// TwinCAT 3 PLC project OC_Profinet
// Title: OC_Profinet
// Company: Open Commissioning
// Author: SpiraTec AG
// ProjectVersion: 1.0.1
// Description: Open Commissioning Library for Profinet devices
// ProgramVersion: 3.1.4026.19
// libraries:
//   OC_Core, * (Open Commissioning)
//   OC_Profisafe, * (Open Commissioning)
//   Tc2_Math, * (Beckhoff Automation GmbH)
//   Tc2_Standard, * (Beckhoff Automation GmbH)
//   Tc2_System, * (Beckhoff Automation GmbH)
//   Tc2_Utilities, * (Beckhoff Automation GmbH)
//   Tc3_Module, * (Beckhoff Automation GmbH)
//   TcUnit, * (www.tcunit.org)
// project tree:
//   Common/ProfidriveGSM/ E_ProfidriveGSM_State.TcTLEO, FB_ProfidriveGSM.TcPOU, ST_ProfidriveGSM_Control.TcDUT, ST_ProfidriveGSM_Status.TcDUT
//   Common/ProfidriveParamInterpreter/ E_ProfidriveParam_Format.TcDUT, FB_ProfidriveParamInterpreter.TcPOU, ST_ProfidriveParam.TcDUT, ST_ProfidriveParam_Set.TcDUT
//   Common/Utils/ F_CalcCrc16.TcPOU
//   Devices/ I_SEW_Movisafe.TcIO
//   Devices/Profidrive_Telegram1/ FB_Profidrive_Telegram1.TcPOU, ST_Profidrive_Telegram1_Config.TcDUT, ST_Profidrive_Telegram1_Control.TcDUT, ST_Profidrive_Telegram1_Status.TcDUT
//   Devices/Siemens_RcvDp/ FB_Siemens_RcvDp.TcPOU, ST_Siemens_RcvDp_Config.TcDUT, ST_Siemens_RcvDp_Control.TcDUT, ST_Siemens_RcvDp_DevData.TcDUT, ST_Siemens_RcvDp_HstData.TcDUT, ST_Siemens_RcvDp_Status.TcDUT
//   Devices/Siemens_SendDp/ FB_Siemens_SendDp.TcPOU, ST_Siemens_SendDp_Config.TcDUT, ST_Siemens_SendDp_Control.TcDUT, ST_Siemens_SendDp_DevData.TcDUT, ST_Siemens_SendDp_HstData.TcDUT, ST_Siemens_SendDp_Status.TcDUT
//   Devices/SEW_MoviC_Position/ E_SEW_MoviC_Position_OperationMode.TcDUT, FB_SEW_MoviC_Position.TcPOU, ST_SEW_MoviC_Position_Config.TcDUT, ST_SEW_MoviC_Position_Control.TcDUT, ST_SEW_MoviC_Position_Status.TcDUT
//   Devices/SEW_MoviC_Velocity/ FB_SEW_MoviC_Velocity.TcPOU, ST_SEW_MoviC_Velocity_Config.TcDUT, ST_SEW_MoviC_Velocity_Control.TcDUT, ST_SEW_MoviC_Velocity_Status.TcDUT
//   Devices/SEW_Movisafe_CSSx1a/ FB_SEW_Movisafe_CSSx1a.TcPOU, ST_SEW_Movisafe_CSSx1a_Config.TcDUT, ST_SEW_Movisafe_CSSx1a_Control.TcDUT, ST_SEW_Movisafe_CSSx1a_Status.TcDUT
//   / PlcTask.TcTTO
//   Tests/Devices/ FB_ProfidriveGSM_Test.TcPOU, FB_ProfidriveTelegram1_Test.TcPOU, FB_SEW_MoviC_Position_Test.TcPOU, FB_SEW_MoviC_Velocity_Test.TcPOU, FB_Siemens_RcvDp_Test.TcPOU, FB_SEW_Movisafe_CSSx1a_Test.TcPOU, FB_Siemens_SendDp_Test.TcPOU
//   Tests/Helpers/ FB_SEW_Movisafe.TcPOU
//   Tests/ PRG_TEST.TcPOU
//   _backlog/Danfoss_VLT_MCA_120/ FB_Danfoss_VLT_MCA_120.TcPOU, ST_Danfoss_VLT_MCA_120_Config.TcDUT, ST_Danfoss_VLT_MCA_120_Control.TcDUT, ST_Danfoss_VLT_MCA_120_Status.TcDUT (not stored)
//   _backlog/ProfidriveCu/ FB_ProfidriveCu.TcPOU, I_Sinamics.TcIO (not stored), ST_ProfidriveCuConfig.TcDUT (not stored)
//   _backlog/SEW_Movisafe_CSBx1a/ FB_SEW_Movisafe_CSBx1a.TcPOU, ST_SEW_Movisafe_CSBx1a_Config.TcDUT, ST_SEW_Movisafe_CSBx1a_Control.TcDUT, ST_SEW_Movisafe_CSBx1a_Status.TcDUT

CONFIGURATION OC_Profinet
    RESOURCE PLC ON TwinCAT3
        TASK PlcTask(INTERVAL := T#1ms, PRIORITY := 6);
        PROGRAM PRG_TEST WITH PlcTask : PRG_TEST;
    END_RESOURCE
END_CONFIGURATION

// ---- Common/ProfidriveGSM/E_ProfidriveGSM_State.TcTLEO
{attribute 'qualified_only'}
{attribute 'strict'}
{attribute 'conditionalshow'}
TYPE E_ProfidriveGSM_State :
(
	S0_Disabled := 0,
	S1_SwitchingOnInhibited := 1,
	S2_ReadyForSwitchingOn := 2,
	S3_SwitchedOn := 3,
	S4_Operation := 4,
	S51_RampStop := 51,
	S52_QuickStop := 52
);
END_TYPE

// ---- Common/ProfidriveGSM/ST_ProfidriveGSM_Control.TcDUT
(*
	Steuerwort 1 (STW1)
	Steuerwort 1 SIEMENS Telegramm 10x
	https://cache.industry.siemens.com/dl/files/665/109770665/att_1023132/v2/109770665_PROFIdrive_Statemachine_DOC_V10_de.pdf
*)
{attribute 'pack_mode' := '1'}
TYPE ST_ProfidriveGSM_Control :
STRUCT
	b0_On 							: BIT; 	//ON/OFF (OFF1)
	b1_CoastStop					: BIT; 	//The axis will not coast stop if this bit is set (OFF2)
	b2_QuickStop					: BIT; 	//The axis will not execute quick stop if this bit is set. Quick stop executes a controlled stop on the axis. (OFF3)
	b3_EnableOperation				: BIT; 	//The axis will enable and execute command if all preconditions are set. If a Wake and Shake procedure has to be executed as part of enabling, the transition to state "S4: Operation Enabled" is delayed until the procedure is finished.
	b4_Reserve						: BIT;	//Reserve
	b5_Reserve						: BIT;	//Reserve
	b6_Reserve						: BIT;	//Reserve
	b7_FaultAcknowledge				: BIT;	//Set this bit to reset faults on the drive.
	b8_Reserve						: BIT;	//Reserve
	b9_Reserve						: BIT;	//Reserve	
	b10_ControlPlc					: BIT;	//When not set, no command is accepted from the PLC.	
	b11_Reserved					: BIT;	//Reserve
	b12_Reserved					: BIT;	//Reserve
	b13_Reserved					: BIT;	//Reserve
	b14_Reserved					: BIT;	//Reserve
	b15_Reserved					: BIT;	//Reserve
END_STRUCT
END_TYPE

// ---- Common/ProfidriveGSM/ST_ProfidriveGSM_Status.TcDUT
(*
	Zustandswort 1 (ZSW1)
	Zustandswort 1 SIEMENS Telegramm 10x
	https://cache.industry.siemens.com/dl/files/665/109770665/att_1023132/v2/109770665_PROFIdrive_Statemachine_DOC_V10_de.pdf
*)

{attribute 'pack_mode' := '1'}
TYPE ST_ProfidriveGSM_Status :
STRUCT
	b0_ReadyToSwitchOn 				: BIT; 	//Ready to switch on
	b1_ReadyForOperation			: BIT; 	//Ready for operation
	b2_OperationEnabled				: BIT; 	//Operation enabled
	b3_FaultPresent					: BIT; 	//A fault is present on the axis
	b4_CoastStop 					: BIT;	//No coast stop is executed (No OFF2 is active)
	b5_QuickStop					: BIT;	//No quick stop is executed (No OFF3 is active)
	b6_SwitchingOnInhibited			: BIT;	//Switch-on inhibit Switching on again is only possible through OFF1 and subsequent ON.
	b7_WarningPresent				: BIT;	//Warning present. The drive is operating. No acknowledgment required
	b8_Reserve						: BIT;	//Reserve
	b9_ControlRequested				: BIT;	//Control requested by the master
	b10_Reserved					: BIT;	//Reserve
	b11_Reserved					: BIT;	//Reserve
	b12_Reserved					: BIT;	//Reserve
	b13_Reserved					: BIT;	//Reserve
	b14_Reserved					: BIT;	//Reserve
	b15_Reserved					: BIT;	//Reserve
END_STRUCT
END_TYPE

// ---- Common/ProfidriveParamInterpreter/E_ProfidriveParam_Format.TcDUT
{attribute 'qualified_only'}
{attribute 'strict'}
{attribute 'conditionalshow'}
TYPE E_ProfidriveParam_Format :
(
	UNKNOWN := 0,
	INT8	:= 2,
	INT16	:= 3,
	INT32	:= 4,
	UINT8	:= 5,
	UINT16	:= 6,
	UINT32	:= 7,
	FLOAT	:= 8,
	ZERO	:= 64,
	BYTE_	:= 65,
	WORD_	:= 66,
	DWORD_	:= 67,
	ERROR	:= 68
) BYTE;
END_TYPE

// ---- Common/ProfidriveParamInterpreter/ST_ProfidriveParam.TcDUT
{attribute 'conditionalshow'}
TYPE ST_ProfidriveParam :
STRUCT
	nAttribute	: BYTE;
	nNumber		: UINT;
	nSubIndex	: UINT;
	nElements	: BYTE;
	nFormat		: E_ProfidriveParam_Format;
	aValue		: ARRAY[0..234] OF BYTE;
END_STRUCT
END_TYPE

// ---- Common/ProfidriveParamInterpreter/ST_ProfidriveParam_Set.TcDUT
{attribute 'conditionalshow'}
TYPE ST_ProfidriveParam_Set :
	ARRAY[0..22] OF ST_ProfidriveParam; 
END_TYPE

// ---- Devices/Profidrive_Telegram1/ST_Profidrive_Telegram1_Config.TcDUT
TYPE ST_Profidrive_Telegram1_Config :
STRUCT
	bForceMode					: BOOL; //Ignore process data from fieldbus.
	bSwapProcessData			: BOOL; //Reverse process data byte order from/to fieldbus.
	fRampDownTimeCoastStop 		: REAL := 1.0;		//Coast stop deceleration time in s
	bControlRequested			: BOOL := TRUE;
	bOutputVelocity				: BOOL := TRUE;		//TRUE: TargetValue = Velocity, FALSE: TargetValue = Position
	fP1058						: REAL := 150.0;	//JOG 1 velocity in rotation/s
	fP1059						: REAL := -150.0;	//JOG 1 velocity in rotation/s
	fP1120						: REAL := 2.0;		//Default acceleration time in s
	fP1121						: REAL := 2.0;		//Default deceleration time in s
	fP1135						: REAL := 1.0;		//Ramp down time quick stop in s
	fP2000						: REAL := 3000;		//Velocity in rotation/s when targeting 16#4000
	nR0035						: REAL := 60.0; 	//Temperature in degree celcius	
END_STRUCT
END_TYPE

// ---- Devices/Profidrive_Telegram1/ST_Profidrive_Telegram1_Control.TcDUT
TYPE ST_Profidrive_Telegram1_Control :
STRUCT
	b0_Off1								: BOOL;	//STW1_0	0 = OFF1 (braking with ramp-function generator, then pulse suppression & ready for switching on) | 0 → 1 = ON (pulses can be enabled)
	b1_Off2								: BOOL;	//STW1_1	0 = OFF2 (immediate pulse suppression and switching on inhibited) | 1 = No OFF2 (enable is possible)
	b2_Off3								: BOOL;	//STW1_2	0 = OFF3 (braking with the OFF3 ramp p1135, then pulse suppression and switching on inhibited) | 1 = No OFF3 (enable possible) 
	b3_EnableOperation					: BOOL;	//STW1_3	0 = Inhibit operation (suppress pulses) | 1 = Enable operation (pulses can be enabled) 
	b4_OperatingCondition				: BOOL;	//STW1_4	0 = Inhibit ramp-function generator (set the ramp-function generator output to zero) | 1 = Operating condition (the ramp-function generator can be enabled)
	b5_ContinueRampFunctionGenerator	: BOOL;	//STW1_5	0 = Freeze ramp-function generator (freeze the ramp-function generator output) | 1 = Continue ramp-function generator 
	b6_EnableSetpoint  					: BOOL;	//STW1_6	0 = Inhibit setpoint (set the ramp-function generator input to zero) | 1 = Enable setpoint 
	b7_AcknowledgeFaults				: BOOL;	//STW1_7	0 → 1: = Acknowledge faults	                            
	b8_Jog1								: BOOL;	//STW1_8	1 = Jog 1 signal source
	b9_Jog2								: BOOL;	//STW1_9	1 = Jog 2 signal source
	b10_ControlByPlc					: BOOL;	//STW1_10	1 = Control by PLC
	b11_SetpointInversion				: BOOL;	//STW1_11	1 = Setpoint inversion
	b12_Reserved						: BOOL;	//STW1_12	Reserved
	b13_PotentiometerSetpointRaise		: BOOL;	//STW1_13	1 = Motorized potentiometer setpoint raise
	b14_PotentiometerSetpointLower		: BOOL;	//STW1_14	1 = Motorized potentiometer setpoint lower
	b15_Reserved						: BOOL;	//STW1_15	Reserved	
	nTargetVelocity						: INT;
END_STRUCT
END_TYPE

// ---- Devices/Profidrive_Telegram1/ST_Profidrive_Telegram1_Status.TcDUT
TYPE ST_Profidrive_Telegram1_Status :
STRUCT
	b0_ReadyForSwitchingOn				: BOOL; // ZSW1_0	1 = Ready for switching on
	b1_ReadyForOperation				: BOOL; // ZSW1_1	1 = Ready for operation
	b2_OperationEnabled					: BOOL; // ZSW1_2	1 = Operation enabled
	b3_FaultPresent						: BOOL; // ZSW1_3	1 = Fault present
	b4_NoCoastDownActive				: BOOL; // ZSW1_4	1 = No coast down active (OFF2 inactive)
	b5_NoQuickStopActive				: BOOL; // ZSW1_5	1 = No quick stop active (OFF3 inactive)
	b6_SwitchingOnInhibited				: BOOL; // ZSW1_6	1 = Switching on inhibited active
	b7_AlarmPresent						: BOOL; // ZSW1_7	1 = Alarm present                        	
	b8_DeviationWithinTolerance			: BOOL; // ZSW1_8	1 = Speed setpoint - actual value deviation within tolerance t_off
	b9_ControlRequested					: BOOL; // ZSW1_9	1 = Control requested        
	b10_RpmCompValueReachedOrExceeded	: BOOL; // ZSW1_10	1 = f or n comparison value reached/exceeded  
	b11_TorqueOrPowerLimitNotReached	: BOOL; // ZSW1_11	1 = I, M, or P limit not reached     
	b12_OpenHoldingBrake 				: BOOL; // ZSW1_12	1 = Open the holding brake      
	b13_NoOvertempAlarm					: BOOL; // ZSW1_13	1 = No motor overtemperature alarm      
	b14_MotorRotatesForwards			: BOOL; // ZSW1_14	1 = Motor rotates forwards (n_act >= 0) | 0 = Motor rotates backwards (n_act < 0)   
	b15_NoAlarmNoOvertempPowerUnit		: BOOL; // ZSW1_15	1 = No alarm, thermal overload, power unit  
	nVelocity							: INT;
END_STRUCT
END_TYPE

// ---- Devices/Siemens_RcvDp/ST_Siemens_RcvDp_Config.TcDUT
TYPE ST_Siemens_RcvDp_Config :
STRUCT
	bForceMode			: BOOL; //Ignore process data from fieldbus.
	bSwapProcessData	: BOOL; //Reverse process data byte order from/to fieldbus.
	nDpDpId			 	: UINT := 0;
	fTimeout		 	: REAL := 0.5;
	bAutoAckRei			: BOOL := TRUE;
END_STRUCT
END_TYPE

// ---- Devices/Siemens_RcvDp/ST_Siemens_RcvDp_Control.TcDUT
{attribute 'pack_mode' := '1'}
TYPE ST_Siemens_RcvDp_Control :
STRUCT
	nRcvBoolData			: WORD;
	nRcvInt00				: INT;
	nRcvInt01				: INT;
	nRcvData				: WORD;
	nRcvSequenceNumber		: WORD;
	nRcvCrc					: WORD;
END_STRUCT
END_TYPE

// ---- Devices/Siemens_RcvDp/ST_Siemens_RcvDp_DevData.TcDUT
TYPE ST_Siemens_RcvDp_DevData :
STRUCT
	bAckRei		: BOOL;
	bSub00		: BOOL;
	bSub01		: BOOL;
	bSub02		: BOOL;
	bSub03		: BOOL;
	bSub04		: BOOL;
	bSub05		: BOOL;
	bSub06		: BOOL;
	bSub07		: BOOL;
	bSub08		: BOOL;
	bSub09		: BOOL;
	bSub10		: BOOL;
	bSub11		: BOOL;
	bSub12		: BOOL;
	bSub13		: BOOL;
	bSub14		: BOOL;
	bSub15		: BOOL;
	nSub00		: INT;
	nSub01		: INT;
END_STRUCT
END_TYPE

// ---- Devices/Siemens_RcvDp/ST_Siemens_RcvDp_HstData.TcDUT
TYPE ST_Siemens_RcvDp_HstData :
STRUCT
	bError		: BOOL;
	bSubsOn		: BOOL;
	bRcv00		: BOOL;
	bRcv01		: BOOL;
	bRcv02		: BOOL;
	bRcv03		: BOOL;
	bRcv04		: BOOL;
	bRcv05		: BOOL;
	bRcv06		: BOOL;
	bRcv07		: BOOL;
	bRcv08		: BOOL;
	bRcv09		: BOOL;
	bRcv10		: BOOL;
	bRcv11		: BOOL;
	bRcv12		: BOOL;
	bRcv13		: BOOL;
	bRcv14		: BOOL;
	bRcv15		: BOOL;
	nRcv00		: INT;
	nRcv01		: INT;
END_STRUCT
END_TYPE

// ---- Devices/Siemens_RcvDp/ST_Siemens_RcvDp_Status.TcDUT
{attribute 'pack_mode' := '1'}
TYPE ST_Siemens_RcvDp_Status :
STRUCT
	nSendData				: WORD;
	nSendSequenceNumber		: WORD;	
	nSendCrc				: WORD;
END_STRUCT
END_TYPE

// ---- Devices/Siemens_SendDp/ST_Siemens_SendDp_Config.TcDUT
TYPE ST_Siemens_SendDp_Config :
STRUCT
	bForceMode			: BOOL; //Ignore process data from fieldbus.
	bSwapProcessData	: BOOL; //Reverse process data byte order from/to fieldbus.
	nDpDpId			 	: UINT := 0;
	fTimeout		 	: REAL := 0.5;
END_STRUCT
END_TYPE

// ---- Devices/Siemens_SendDp/ST_Siemens_SendDp_Control.TcDUT
TYPE ST_Siemens_SendDp_Control :
STRUCT
	nRcvData				: WORD;
	nRcvSequenceNumber		: WORD;	
	nRcvCrc					: WORD;
END_STRUCT
END_TYPE

// ---- Devices/Siemens_SendDp/ST_Siemens_SendDp_DevData.TcDUT
TYPE ST_Siemens_SendDp_DevData :
STRUCT
	bSend00		: BOOL;
	bSend01		: BOOL;
	bSend02		: BOOL;
	bSend03		: BOOL;
	bSend04		: BOOL;
	bSend05		: BOOL;
	bSend06		: BOOL;
	bSend07		: BOOL;
	bSend08		: BOOL;
	bSend09		: BOOL;
	bSend10		: BOOL;
	bSend11		: BOOL;
	bSend12		: BOOL;
	bSend13		: BOOL;
	bSend14		: BOOL;
	bSend15		: BOOL;
	nSend00		: INT;
	nSend01		: INT;
END_STRUCT
END_TYPE

// ---- Devices/Siemens_SendDp/ST_Siemens_SendDp_HstData.TcDUT
TYPE ST_Siemens_SendDp_HstData :
STRUCT
	bError		: BOOL;
	bSubsOn		: BOOL;
END_STRUCT
END_TYPE

// ---- Devices/Siemens_SendDp/ST_Siemens_SendDp_Status.TcDUT
TYPE ST_Siemens_SendDp_Status :
STRUCT
	nSendBoolData			: WORD;
	nSendInt00				: INT;
	nSendInt01				: INT;
	nSendData				: WORD;
	nSendSequenceNumber		: WORD;
	nSendCrc				: WORD;
END_STRUCT
END_TYPE

// ---- Devices/SEW_MoviC_Position/E_SEW_MoviC_Position_OperationMode.TcDUT
{attribute 'qualified_only'}
TYPE E_SEW_MoviC_Position_OperationMode :
(
	Jog					:= 100, //Position controlled jogging
	JogNoEnc			:= 101, //Speed controlled jogging
	SpeedControl		:= 200, //Speed control
	ReferenceParam		:= 300, //Reference travel, offset via parameter
	ReferenceBus		:= 301, //Reference travel, offset via fieldbus
	PositionAbs			:= 400, //Absolute position control
	PositionRel			:= 401, //Relative position control
	PositionModPos		:= 402, //Modulo position control, positive
	PositionModNeg		:= 403, //Modulo position control, negative
	PositionModShort	:= 404, //Modulo position control, shortest distance
	EnergyOptimized		:= 1200, //Energieoptimiertes Positionieren
	MechanicsOptimized	:= 1210	 //Mechanikoptimiertes Positionieren
)INT;
END_TYPE

// ---- Devices/SEW_MoviC_Position/ST_SEW_MoviC_Position_Config.TcDUT
TYPE ST_SEW_MoviC_Position_Config :
STRUCT
	bForceMode				: BOOL; //Ignore process data from fieldbus.
	bSwapProcessData		: BOOL; //Reverse process data byte order from/to fieldbus.
	nSoftwareLimitMin		: DINT := -2147483648;	//Position limit minimum in LU
	nSoftwareLimitMax		: DINT := 2147483647;	//Position limit maximum in LU
	nReferencePos			: DINT := 0;			//Reference position in LU when using mode 300
	fDecCoastStop			: REAL := 1000.0;		//Deceleration for coast/brake stop in LU/s^2
	fDecEstop				: REAL := 100.0;		//Deceleration for emergency stop in LU/s^2
	fDecelerationLimit		: REAL := 100.0;		//Decceleration limit (bus stop) in LU/s^2
	fRatioVelocity			: REAL := 1.0;			//Ratio for setpoint velocity
	fRatioAccDec			: REAL := 1.0;			//Ratio for setpoint acceleration/deceleration
	fRatioPosition			: REAL := 1.0;			//Ratio for position output
	nJerk					: INT  := 0;			//Jerk from 0 to 100%
	fPositionOffset			: REAL := 0;
	fInitPosition			: REAL := 0;
	fResolution				: REAL := 0.1;
END_STRUCT
END_TYPE

// ---- Devices/SEW_MoviC_Position/ST_SEW_MoviC_Position_Control.TcDUT
{attribute 'pack_mode' := '1'}
TYPE ST_SEW_MoviC_Position_Control :
STRUCT
    b0_EnableEStop 					: BIT;	//0  1 = enable, 0 = emergency stop
    b1_EnableBusStop 				: BIT;	//1  1 = enable, 0 = stop at application limits
    b2_Reserved2 					: BIT;	//2
    b3_ReleaseBrake 				: BIT;	//3  only needed if function is activated
    b4_JoggingCW 					: BIT;	//4  jog positive
    b5_JoggingCCW 					: BIT;	//5  jog negative
    b6_AcceptRelativePosition 		: BIT;	//6  apply relative target pos only in relative pos mode
    b7_StartStop 					: BIT;	//7  1 = start movement in all modes except jog, 0 = deceleration to speed 0
    b8_ErrorReset 					: BIT;	//8  reset fault messages
    b9_Reserved9 					: BIT;	//9
    b10_ActivateDriveTrain2 		: BIT;	//10  0 = drive train 1 selected, 1 = drive train 2 selected
    b11_Reserved11 					: BIT;	//11
    b12_DisableSoftwareLimits 		: BIT;	//12  0 = software limit activated, 1 = software limit deactivated
    b13_ActivateInhibit 			: BIT;	//13  1 = output stage inhibit activated -> motor coasts to halt or brake is applied, 0 = output stage can be enabled
    b14_ActivateStandByMode 		: BIT;	//14  1 = activated, can only be activated when output stage is inhibited (bActivateInhibit = 1)
    b15_MovikitHeartbeat 			: BIT;	//15  Heartbeat trigger
	nSetpointSpeed					: INT;	//16..31 
	nSetpointAcceleration			: INT;	//32..47
	nSetpointDeceleration			: INT;	//48..63
	nDigitalOutputs					: WORD;	//64..79
	nTargetApplicationMode			: E_SEW_MoviC_Position_OperationMode; //80..95
	nTargetPosition					: DINT;	//96..127
END_STRUCT
END_TYPE

// ---- Devices/SEW_MoviC_Position/ST_SEW_MoviC_Position_Status.TcDUT
{attribute 'pack_mode' := '1'}
TYPE ST_SEW_MoviC_Position_Status :
STRUCT
	b0_InverterReady					: BIT;	//0  1 = Ready
	b1_STOInactive						: BIT;	//1  1 = STO inactive
	b2_PowerStageOn						: BIT;	//2  1 = Output stage enable
	b3_BrakeReleased					: BIT;	//3  1 = Brake released
	b4_MotorTurning						: BIT;	//4  1 = Motor running
	b5_DriveReferenced					: BIT;	//5  1 = Active drive referenced
	b6_SetpointsActive					: BIT;	//6  1 = New relative position applied
	b7_TargetpositionReached			: BIT;	//7  1 = In position
	b8_ErrorActive						: BIT;	//8  1 = Fault
	b9_WarningActive					: BIT;	//9  1 = Warning
	b10_DriveTrain2Active				: BIT;	//10  1 = Drive train 2 active
	b11_SpeedSetpointReached			: BIT;	//11  1 = "Setpoint/actual speed comparison active" signal
	b12_SoftwareLimitsDisabled			: BIT;	//12  1 = Software limit switches inactive
	b13_OutputStageInhibit 				: BIT;	//13  1 = Output stage inhibit 
	b14_StandByModeActive				: BIT;	//14  1 = Standby mode active
	b15_MovikitHeartbeat				: BIT;	//15  Heartbeat trigger mirror
	nActualSpeed						: INT;	//16..31
	nActualStatus						: WORD;	//32..47
	nActualTorque						: INT;	//48..63
	nDigitalInputs						: WORD;	//64..79
	nActualApplicationMode				: E_SEW_MoviC_Position_OperationMode; //80..95
	nActualPosition						: DINT;	//96..127 
END_STRUCT
END_TYPE

// ---- Devices/SEW_MoviC_Velocity/ST_SEW_MoviC_Velocity_Config.TcDUT
TYPE ST_SEW_MoviC_Velocity_Config :
STRUCT
	bForceMode				: BOOL; //Ignore process data from fieldbus.
	bSwapProcessData		: BOOL; //Reverse process data byte order from/to fieldbus.
	nSoftwareLimitMin		: DINT := -2147483648;	//Position limit minimum in LU
	nSoftwareLimitMax		: DINT := 2147483647;	//Position limit maximum in LU
	nReferencePos			: DINT := 0;			//Reference position in LU when using mode 300
	fDecCoastStop			: REAL := 1000.0;		//Deceleration for coast/brake stop in LU/s^2
	fDecEstop				: REAL := 100.0;		//Deceleration for emergency stop in LU/s^2
	fDecelerationLimit		: REAL := 100.0;		//Decceleration limit (bus stop) in LU/s^2
	fRatioVelocity			: REAL := 1.0;			//Ratio for setpoint velocity
	fRatioAccDec			: REAL := 1.0;			//Ratio for setpoint acceleration/deceleration
	fRatioPosition			: REAL := 1.0;			//Ratio for position output
	nJerk					: INT  := 0;			//Jerk from 0 to 100%
	fPositionOffset			: REAL := 0;
	fInitPosition			: REAL := 0;
	fResolution				: REAL := 0.1;
	bOutputVelocity			: BOOL := TRUE;			//TRUE: TargetValue = Velocity, FALSE: TargetValue = Position
END_STRUCT
END_TYPE

// ---- Devices/SEW_MoviC_Velocity/ST_SEW_MoviC_Velocity_Control.TcDUT
TYPE ST_SEW_MoviC_Velocity_Control :
STRUCT
    b0_EnableEStop 					: BIT;	//0  1 = enable, 0 = emergency stop
    b1_EnableBusStop 				: BIT;	//1  1 = enable, 0 = stop at application limits
    b2_Reserved2 					: BIT;	//2
    b3_ReleaseBrake 				: BIT;	//3  only needed if function is activated
    b4_JoggingCW 					: BIT;	//4  jog positive
    b5_JoggingCCW 					: BIT;	//5  jog negative
    b6_AcceptRelativePosition 		: BIT;	//6  apply relative target pos only in relative pos mode
    b7_StartStop 					: BIT;	//7  1 = start movement in all modes except jog, 0 = deceleration to speed 0
    b8_ErrorReset 					: BIT;	//8  reset fault messages
    b9_Reserved9 					: BIT;	//9
    b10_ActivateDriveTrain2 		: BIT;	//10  0 = drive train 1 selected, 1 = drive train 2 selected
    b11_Reserved11 					: BIT;	//11
    b12_DisableSoftwareLimits 		: BIT;	//12  0 = software limit activated, 1 = software limit deactivated
    b13_ActivateInhibit 			: BIT;	//13  1 = output stage inhibit activated -> motor coasts to halt or brake is applied, 0 = output stage can be enabled
    b14_ActivateStandByMode 		: BIT;	//14  1 = activated, can only be activated when output stage is inhibited (bActivateInhibit = 1)
    b15_MovikitHeartbeat 			: BIT;	//15  Heartbeat trigger
	nSetpointSpeed					: INT;	//16..31 
	nSetpointAcceleration			: INT;	//32..47
	nSetpointDeceleration			: INT;	//48..63
	nDigitalOutputs					: WORD;	//64..79	
END_STRUCT
END_TYPE

// ---- Devices/SEW_MoviC_Velocity/ST_SEW_MoviC_Velocity_Status.TcDUT
{attribute 'pack_mode' := '1'}
TYPE ST_SEW_MoviC_Velocity_Status :
STRUCT
	b0_InverterReady					: BIT;	//0  1 = Ready
	b1_STOInactive						: BIT;	//1  1 = STO inactive
	b2_PowerStageOn						: BIT;	//2  1 = Output stage enable
	b3_BrakeReleased					: BIT;	//3  1 = Brake released
	b4_MotorTurning						: BIT;	//4  1 = Motor running
	b5_DriveReferenced					: BIT;	//5  1 = Active drive referenced
	b6_SetpointsActive					: BIT;	//6  1 = New relative position applied
	b7_TargetpositionReached			: BIT;	//7  1 = In position
	b8_ErrorActive						: BIT;	//8  1 = Fault
	b9_WarningActive					: BIT;	//9  1 = Warning
	b10_DriveTrain2Active				: BIT;	//10  1 = Drive train 2 active
	b11_SpeedSetpointReached			: BIT;	//11  1 = "Setpoint/actual speed comparison active" signal
	b12_SoftwareLimitsDisabled			: BIT;	//12  1 = Software limit switches inactive
	b13_OutputStageInhibit 				: BIT;	//13  1 = Output stage inhibit 
	b14_StandByModeActive				: BIT;	//14  1 = Standby mode active
	b15_MovikitHeartbeat				: BIT;	//15  Heartbeat trigger mirror
	nActualSpeed						: INT;	//16..31
	nActualStatus						: WORD;	//32..47
	nActualTorque						: INT;	//48..63
	nDigitalInputs						: WORD;	//64..79	
END_STRUCT
END_TYPE

// ---- Devices/SEW_Movisafe_CSSx1a/ST_SEW_Movisafe_CSSx1a_Config.TcDUT
TYPE ST_SEW_Movisafe_CSSx1a_Config :
STRUCT	
	bForceMode			: BOOL; //Ignore process data from fieldbus.
	bSwapProcessData	: BOOL; //Reverse process data byte order from/to fieldbus.
END_STRUCT
END_TYPE

// ---- Devices/SEW_Movisafe_CSSx1a/ST_SEW_Movisafe_CSSx1a_Control.TcDUT
{attribute 'pack_mode' := '1'}
TYPE ST_SEW_Movisafe_CSSx1a_Control :
STRUCT
	b0_0_STO			: BIT; //0.0  Sicher abgeschaltetes Drehmoment
	b0_1_SLI			: BIT; //0.1  Freigabe SLI (Sicher begrenztes Schrittmaß)
	b0_2_SBT			: BIT; //0.2  Freigabe SBT (Sicherer Bremsentest)
	b0_3_Reserved		: BIT; //0.3  Reserve
	b0_4_MutingEncErr	: BIT; //0.4  Muting Geber anwählen
	b0_5_TestModeActice	: BIT; //0.5  Test Modus der Antriebssicherheitsfunktion anwählen
	b0_6_AckFDI			: BIT; //0.6  Quittierung der verriegelten Digitaleingänge
	b0_7_AckError		: BIT; //0.7  Quittierung der Fehler Sicherheitskarte
	b1_0_F_DO0			: BIT; //1.0  F-DO 00 Digitaler Ausgang 0
	b1_1_F_DO1			: BIT; //1.1  F-DO 01 Digitaler Ausgang 1
	b1_2_Reserved		: BIT; //1.2  Reserve
	b1_3_Reserved		: BIT; //1.3  Reserve
	b1_4_Reserved		: BIT; //1.4  Reserve
	b1_5_Reserved		: BIT; //1.5  Reserve
	b1_6_Reserved		: BIT; //1.6  Reserve
	b1_7_Reserved		: BIT; //1.7  Reserve
	b2_0_SOS1			: BIT; //2.0  SOS1 deaktivieren (Sicherer Betriebshalt)
	b2_1_Reserved		: BIT; //2.1  Reserve
	b2_2_SSx1			: BIT; //2.2  Antriebssicherheitsfunktion SSx1 deaktivieren
	b2_3_SSx2			: BIT; //2.3  Antriebssicherheitsfunktion SSx2 deaktivieren
	b2_4_SDI1			: BIT; //2.4  SDI 1 deaktivieren (Sichere Bewegungsrichtung)
	b2_5_SDI2			: BIT; //2.5  SDI 2 deaktivieren (Sichere Bewegungsrichtung)
	b2_6_SLI1			: BIT; //2.6  SLI 1 deaktivieren (Sicher begrenztes Schrittmaß)
	b2_7_SLI2			: BIT; //2.7  SLI 2 deaktivieren (Sicher begrenztes Schrittmaß)
	b3_0_SLS1			: BIT; //3.0  SLS 1 deaktivieren (Sicher begrenzte Geschwindigkeit)
	b3_1_SLS2			: BIT; //3.1  SLS 2 deaktivieren (Sicher begrenzte Geschwindigkeit)
	b3_2_SLS3			: BIT; //3.2  SLS 3 deaktivieren (Sicher begrenzte Geschwindigkeit)
	b3_3_SLS4			: BIT; //3.3  SLS 4 deaktivieren (Sicher begrenzte Geschwindigkeit)
	b3_4_SSR1			: BIT; //3.4  SSR 1 deaktivieren (Sicherer Geschwindigkeitsbereich)
	b3_5_SSR2			: BIT; //3.5  SSR 2 deaktivieren (Sicherer Geschwindigkeitsbereich)
	b3_6_Reserved		: BIT; //3.6  Reserve
	b3_7_Reserved		: BIT; //3.7  Reserve
	b4_0_SLA1			: BIT; //4.0  SLA 1 deaktivieren (Sicher begrenzte Beschleunigung)
	b4_1_SLA2			: BIT; //4.1  SLA 2 deaktivieren (Sicher begrenzte Beschleunigung)
	b4_2_Reserved		: BIT; //4.2  Reserve
	b4_3_Reserved		: BIT; //4.3  Reserve
	b4_4_Reserved		: BIT; //4.4  Reserve
	b4_5_Reserved		: BIT; //4.5  Reserve
	b4_6_Reserved		: BIT; //4.6  Reserve
	b4_7_Reserved		: BIT; //4.7  Reserve
END_STRUCT
END_TYPE

// ---- Devices/SEW_Movisafe_CSSx1a/ST_SEW_Movisafe_CSSx1a_Status.TcDUT
{attribute 'pack_mode' := '1'}
TYPE ST_SEW_Movisafe_CSSx1a_Status :
STRUCT
	b0_0_STOActive		: BIT; //0.0  Sicher abgeschaltetes Drehmoment
	b0_1_ASFDiag		: BIT; //0.1  Mindestens eine Antriebssicherheitsfunktion hat eine Grenze überschritten
	b0_2_SBTActive		: BIT; //0.2  Bremsentest ist aktiv
	b0_3_InputDataValid	: BIT; //0.3  Alle Prozesswerte der F-DI enthalten aktuelle Werte
	b0_4_MutingEncErr	: BIT; //0.4  Geber Muting Funktion ist aktive
	b0_5_TestModeActive	: BIT; //0.5  Test Modus der Antriebssicherheitsfunktion ist aktive
	b0_6_Warning		: BIT; //0.6  Warnung in der Safety-option
	b0_7_ErrorState		: BIT; //0.7  Fehler in der Safety-option
	b1_0_F_DI0			: BIT; //1.0  Zustand digitaler Eingang 1
	b1_1_F_DI1			: BIT; //1.1  Zustand digitaler Eingang 2
	b1_2_F_DI2			: BIT; //1.2  Zustand digitaler Eingang 3
	b1_3_F_DI3			: BIT; //1.3  Zustand digitaler Eingang 4
	b1_4_Reserved		: BIT; //1.4  Reserve
	b1_5_Reserved		: BIT; //1.5  Reserve
	b1_6_Reserved		: BIT; //1.6  Reserve
	b1_7_Reserved		: BIT; //1.7  Reserve
	b2_0_SOS1			: BIT; //2.0  SOS1 ist aktiviert (Sicherer Betriebshalt)
	b2_1_Reserved		: BIT; //2.1  Reserve
	b2_2_SSx1			: BIT; //2.2  SSx1  ist aktiviert
	b2_3_SSx2			: BIT; //2.3  SSx2 ist aktiviert
	b2_4_SDI1			: BIT; //2.4  SDI 1  ist aktiviert (Sichere Bewegungsrichtung)
	b2_5_SDI2			: BIT; //2.5  SDI 2  ist aktiviert (Sichere Bewegungsrichtung)
	b2_6_SLI1			: BIT; //2.6  SLI 1  ist aktiviert (Sicher begrenztes Schrittmaß)
	b2_7_SLI2			: BIT; //2.7  SLI 2  ist aktiviert (Sicher begrenztes Schrittmaß)
	b3_0_SLS1			: BIT; //3.0  SLS 1  ist aktiviert (Sicher begrenzte Geschwindigkeit)
	b3_1_SLS2			: BIT; //3.1  SLS 2  ist aktiviert (Sicher begrenzte Geschwindigkeit)
	b3_2_SLS3			: BIT; //3.2  SLS 3  ist aktiviert (Sicher begrenzte Geschwindigkeit)
	b3_3_SLS4			: BIT; //3.3  SLS 4  ist aktiviert (Sicher begrenzte Geschwindigkeit)
	b3_4_SSR1			: BIT; //3.4  SSR 1  ist aktiviert (Sicherer Geschwindigkeitsbereich)
	b3_5_SSR2			: BIT; //3.5  SSR 2  ist aktiviert (Sicherer Geschwindigkeitsbereich)
	b3_6_Reserved		: BIT; //3.6  Reserve
	b3_7_Reserved		: BIT; //3.7  Reserve
	b4_0_SLA1			: BIT; //4.0  SLA 1  ist aktiviert (Sicher begrenzte Beschleunigung)
	b4_1_SLA2			: BIT; //4.1  SLA 2  ist aktiviert (Sicher begrenzte Beschleunigung)
	b4_2_SSM1			: BIT; //4.2  SSM 1  ist aktiviert (Sichere Geschwindigkeitsüberwachung)
	b4_3_SSM2			: BIT; //4.3  SSM 2  ist aktiviert (Sichere Geschwindigkeitsüberwachung)
	b4_4_SSM3			: BIT; //4.4  SSM 3  ist aktiviert (Sichere Geschwindigkeitsüberwachung)
	b4_5_SSM4			: BIT; //4.5  SSM 4  ist aktiviert (Sichere Geschwindigkeitsüberwachung)
	b4_6_Reserved		: BIT; //4.6  Reserve
	b4_7_Reserved		: BIT; //4.7  Reserve
	b5_0_Reserved		: BIT; //5.0  Reserve
	b5_1_Reserved		: BIT; //5.1  Reserve
	b5_2_Reserved		: BIT; //5.2  Reserve
	b5_3_Reserved		: BIT; //5.3  Reserve
	b5_4_Reserved		: BIT; //5.4  Reserve
	b5_5_Reserved		: BIT; //5.5  Reserve
	b5_6_Reserved		: BIT; //5.6  Reserve
	b5_7_Reserved		: BIT; //5.7  Reserve
END_STRUCT
END_TYPE

// ---- _backlog/Danfoss_VLT_MCA_120/ST_Danfoss_VLT_MCA_120_Config.TcDUT
TYPE ST_Danfoss_VLT_MCA_120_Config :
STRUCT
	fRampDownTimeCoastStop 		: REAL := 1.0;		//Coast stop deceleration time in s
	bControlRequested			: BOOL := TRUE;
	bOutputVelocity				: BOOL := TRUE;		//TRUE: TargetValue = Velocity, FALSE: TargetValue = Position
	fP1058						: REAL := 150.0;	//JOG 1 velocity in rotation/s
	fP1059						: REAL := -150.0;	//JOG 1 velocity in rotation/s
	fP1120						: REAL := 2.0;		//Default acceleration time in s
	fP1121						: REAL := 2.0;		//Default deceleration time in s
	fP1135						: REAL := 1.0;		//Ramp down time quick stop in s
	fP2000						: REAL := 3000;		//Velocity in rotation/s when targeting 16#4000
	nR0035						: REAL := 60.0; 	//Temperature in degree celcius	
	bSwapProcessData			: BOOL; //SWAP Process Data from/to FIELDBUS
END_STRUCT
END_TYPE

// ---- _backlog/Danfoss_VLT_MCA_120/ST_Danfoss_VLT_MCA_120_Control.TcDUT
TYPE ST_Danfoss_VLT_MCA_120_Control :
STRUCT
	bOFF1								: BOOL;	//STW1_0	0 = OFF1 (braking with ramp-function generator, then pulse suppression & ready for switching on) | 0 → 1 = ON (pulses can be enabled)
	bOFF2								: BOOL;	//STW1_1	0 = OFF2 (immediate pulse suppression and switching on inhibited) | 1 = No OFF2 (enable is possible)
	bOFF3								: BOOL;	//STW1_2	0 = OFF3 (braking with the OFF3 ramp p1135, then pulse suppression and switching on inhibited) | 1 = No OFF3 (enable possible) 
	bEnableOperation					: BOOL;	//STW1_3	0 = Inhibit operation (suppress pulses) | 1 = Enable operation (pulses can be enabled) 
	bOperatingCondition					: BOOL;	//STW1_4	0 = Inhibit ramp-function generator (set the ramp-function generator output to zero) | 1 = Operating condition (the ramp-function generator can be enabled)
	bContinueRampFunctionGenerator		: BOOL;	//STW1_5	0 = Freeze ramp-function generator (freeze the ramp-function generator output) | 1 = Continue ramp-function generator 
	bEnableSetpoint  					: BOOL;	//STW1_6	0 = Inhibit setpoint (set the ramp-function generator input to zero) | 1 = Enable setpoint 
	bAcknowledgeFaults					: BOOL;	//STW1_7	0 → 1: = Acknowledge faults	                            
	bJog1								: BOOL;	//STW1_8	1 = Jog 1 signal source
	bJog2								: BOOL;	//STW1_9	1 = Jog 2 signal source
	bDataValid							: BOOL;	//STW1_10	1 = Data Valid
	bFreqCorrDown						: BOOL;	//STW1_11	1 = Frequency correction Down
	bFreqCorrUp							: BOOL;	//STW1_12	1 = Frequency correction Up
	bParameterSelectionLSB				: BOOL;	//STW1_13	1 = Parameter Selection LSB
	bParameterSelectionMSB				: BOOL;	//STW1_14	1 = Parameter Selection MSB
	bReversing							: BOOL;	//STW1_15	1 = Reversing	
	nSoll 								: INT;
END_STRUCT
END_TYPE

// ---- _backlog/SEW_Movisafe_CSBx1a/ST_SEW_Movisafe_CSBx1a_Config.TcDUT
TYPE ST_SEW_Movisafe_CSBx1a_Config :
STRUCT	
	bForceMode			: BOOL; //Ignore process data from fieldbus.
	bSwapProcessData	: BOOL; //Reverse process data byte order from/to fieldbus.
END_STRUCT
END_TYPE

// ---- _backlog/SEW_Movisafe_CSBx1a/ST_SEW_Movisafe_CSBx1a_Control.TcDUT
{attribute 'pack_mode' := '1'}
TYPE ST_SEW_Movisafe_CSBx1a_Control :
STRUCT
	b0_0_STO			: BIT; //0.0 Sicher abgeschaltetes Drehmoment
	b0_1_Reserved		: BIT; //0.1 Reserve
	b0_2_Reserved		: BIT; //0.2 Reserve
	b0_3_Reserved		: BIT; //0.3 Reserve
	b0_4_Reserved		: BIT; //0.4 Reserve
	b0_5_Reserved		: BIT; //0.5 Reserve
	b0_6_AckFDI			: BIT; //0.6 Quittierung der verriegelten Digitaleingänge
	b0_7_AckError		: BIT; //0.7 Quittierung der Fehler Sicherheitskarte
	b1_0_Reserved		: BIT; //1.0 Reserve
	b1_1_Reserved		: BIT; //1.1 Reserve
	b1_2_Reserved		: BIT; //1.2 Reserve
	b1_3_Reserved		: BIT; //1.3 Reserve
	b1_4_Reserved		: BIT; //1.4 Reserve
	b1_5_Reserved		: BIT; //1.5 Reserve
	b1_6_Reserved		: BIT; //1.6 Reserve
	b1_7_Reserved		: BIT; //1.7 Reserve
	b2_0_Reserved		: BIT; //2.0 Reserve
	b2_1_Reserved		: BIT; //2.1 Reserve
	b2_2_SSx1			: BIT; //2.2 Antriebssicherheitsfunktion SSx1 deaktivieren
	b2_3_SSx2			: BIT; //2.3 Antriebssicherheitsfunktion SSx2 deaktivieren
	b2_4_Reserved		: BIT; //2.4 Reserve
	b2_5_Reserved		: BIT; //2.5 Reserve
	b2_6_Reserved		: BIT; //2.6 Reserve
	b2_7_Reserved		: BIT; //2.7 Reserve
END_STRUCT
END_TYPE

// ---- _backlog/SEW_Movisafe_CSBx1a/ST_SEW_Movisafe_CSBx1a_Status.TcDUT
{attribute 'pack_mode' := '1'}
TYPE ST_SEW_Movisafe_CSBx1a_Status :
STRUCT
	b0_0_StoActive		: BIT; //0.0 Sicher abgeschaltetes Drehmoment
	b0_1_Reserved		: BIT; //0.1 Reserve
	b0_2_Reserved		: BIT; //0.2 Reserve
	b0_3_InputDataValid	: BIT; //0.3 Alle Prozesswerte der F-DI enthalten aktuelle Werte
	b0_4_Reserved		: BIT; //0.4 Reserve
	b0_5_Reserved		: BIT; //0.5 Reserve
	b0_6_Warning		: BIT; //0.6 Warnung in der Safety-option
	b0_7_ErrorState		: BIT; //0.7 Fehler in der Safety-option
	b1_0_F_DI0			: BIT; //1.0 Zustand digitaler Eingang 1
	b1_1_F_DI1			: BIT; //1.1 Zustand digitaler Eingang 2
	b1_2_F_DI2			: BIT; //1.2 Zustand digitaler Eingang 3
	b1_3_F_DI3			: BIT; //1.3 Zustand digitaler Eingang 4
	b1_4_Reserved		: BIT; //1.4 Reserve
	b1_5_Reserved		: BIT; //1.5 Reserve
	b1_6_Reserved		: BIT; //1.6 Reserve
	b1_7_Reserved		: BIT; //1.7 Reserve
	b2_0_Reserved		: BIT; //2.0 Reserve
	b2_1_Reserved		: BIT; //2.1 Reserve
	b2_2_SSx1			: BIT; //2.2 SSx1  ist aktiviert
	b2_3_SSx2			: BIT; //2.3 SSx2 ist aktiviert
	b2_4_Reserved		: BIT; //2.4 Reserve
	b2_5_Reserved		: BIT; //2.5 Reserve
	b2_6_Reserved		: BIT; //2.6 Reserve
	b2_7_Reserved		: BIT; //2.7 Reserve
	b3_0_Reserved		: BIT; //3.0 Reserve
	b3_1_Reserved		: BIT; //3.1 Reserve
	b3_2_Reserved		: BIT; //3.2 Reserve
	b3_3_Reserved		: BIT; //3.3 Reserve
	b3_4_Reserved		: BIT; //3.4 Reserve
	b3_5_Reserved		: BIT; //3.5 Reserve
	b3_6_Reserved		: BIT; //3.6 Reserve
	b3_7_Reserved		: BIT; //3.7 Reserve
END_STRUCT
END_TYPE

// ---- Devices/I_SEW_Movisafe.TcIO
INTERFACE I_SEW_Movisafe

PROPERTY bSTO : BOOL
GET
END_GET
END_PROPERTY

END_INTERFACE

// ---- Tests/PRG_TEST.TcPOU
PROGRAM PRG_TEST
VAR
	FB_ProfidriveGSM_Test : FB_ProfidriveGSM_Test;
	FB_ProfidriveTelegram1_Test : FB_ProfidriveTelegram1_Test;
	FB_SEW_MoviC_Position_Test :FB_SEW_MoviC_Position_Test;
	FB_SEW_MoviC_Velocity_Test : FB_SEW_MoviC_Velocity_Test;
	FB_SEW_Movisafe_CSSx1a_Test : FB_SEW_Movisafe_CSSx1a_Test;
	FB_Siemens_RcvDp_Test : FB_Siemens_RcvDp_Test;
	FB_Siemens_SendDp_Test : FB_Siemens_SendDp_Test;
	
	fbSystem : FB_System;
END_VAR

fbSystem();
TcUnit.RUN();

END_PROGRAM

// ---- Tests/Devices/FB_ProfidriveGSM_Test.TcPOU
FUNCTION_BLOCK FB_ProfidriveGSM_Test EXTENDS TcUnit.FB_TestSuite

TestState_S0();
TestState_S1();
TestState_S2();
TestState_S3();
TestState_S4();
TestState_S51();
TestState_S52();

TestTransitions_S0();
TestTransitions_S1();
TestTransitions_S2();
TestTransitions_S3();
TestTransitions_S4();
TestTransitions_S51();
TestTransitions_S52();

METHOD TestState_S0 : BOOL
VAR
	fbFSM 				: FB_ProfidriveGSM;
	stStatusExpected	: ST_ProfidriveGSM_Status;
END_VAR
TEST('Set State S0');

//Arrange
fbFSM.eState := E_ProfidriveGSM_State.S0_Disabled;

stStatusExpected.b0_ReadyToSwitchOn 		:= FALSE;				
stStatusExpected.b1_ReadyForOperation 		:= FALSE;				
stStatusExpected.b2_OperationEnabled 		:= FALSE;
stStatusExpected.b6_SwitchingOnInhibited 	:= FALSE;

//Act
fbFSM();

//Assert

AssertEquals_BOOL(stStatusExpected.b0_ReadyToSwitchOn, fbFSM.nStatus.b0_ReadyToSwitchOn, 'b0_ReadyToSwitchOn: AssertEquals not returning expected value');
AssertEquals_BOOL(stStatusExpected.b1_ReadyForOperation, fbFSM.nStatus.b1_ReadyForOperation, 'b1_ReadyForOperation: AssertEquals not returning expected value');
AssertEquals_BOOL(stStatusExpected.b2_OperationEnabled, fbFSM.nStatus.b2_OperationEnabled, 'b2_OperationEnabled: AssertEquals not returning expected value');	
AssertEquals_BOOL(stStatusExpected.b6_SwitchingOnInhibited, fbFSM.nStatus.b6_SwitchingOnInhibited, 'b6_SwitchingOnInhibited: AssertEquals not returning expected value');	

TEST_FINISHED();
END_METHOD

METHOD TestState_S1 : BOOL
VAR
	fbFSM 				: FB_ProfidriveGSM;
	stStatusExpected	: ST_ProfidriveGSM_Status;
END_VAR
TEST('Set State S1');

//Arrange
fbFSM.eState := E_ProfidriveGSM_State.S1_SwitchingOnInhibited;

stStatusExpected.b0_ReadyToSwitchOn 		:= FALSE;				
stStatusExpected.b1_ReadyForOperation 		:= FALSE;				
stStatusExpected.b2_OperationEnabled 		:= FALSE;
stStatusExpected.b6_SwitchingOnInhibited 	:= TRUE;

//Act
fbFSM();

//Assert
AssertEquals_BOOL(stStatusExpected.b0_ReadyToSwitchOn, fbFSM.nStatus.b0_ReadyToSwitchOn, 'b0_ReadyToSwitchOn: AssertEquals not returning expected value');
AssertEquals_BOOL(stStatusExpected.b1_ReadyForOperation, fbFSM.nStatus.b1_ReadyForOperation, 'b1_ReadyForOperation: AssertEquals not returning expected value');
AssertEquals_BOOL(stStatusExpected.b2_OperationEnabled, fbFSM.nStatus.b2_OperationEnabled, 'b2_OperationEnabled: AssertEquals not returning expected value');	
AssertEquals_BOOL(stStatusExpected.b6_SwitchingOnInhibited, fbFSM.nStatus.b6_SwitchingOnInhibited, 'b6_SwitchingOnInhibited: AssertEquals not returning expected value');	

TEST_FINISHED();
END_METHOD

METHOD TestState_S2 : BOOL
VAR
	fbFSM 				: FB_ProfidriveGSM;
	stStatusExpected	: ST_ProfidriveGSM_Status;
END_VAR
TEST('Set State S2');

//Arrange
fbFSM.eState := E_ProfidriveGSM_State.S2_ReadyForSwitchingOn;

stStatusExpected.b0_ReadyToSwitchOn 		:= TRUE;				
stStatusExpected.b1_ReadyForOperation 		:= FALSE;				
stStatusExpected.b2_OperationEnabled 		:= FALSE;
stStatusExpected.b6_SwitchingOnInhibited 	:= FALSE;

//Act
fbFSM();

//Assert
AssertEquals_BOOL(stStatusExpected.b0_ReadyToSwitchOn, fbFSM.nStatus.b0_ReadyToSwitchOn, 'b0_ReadyToSwitchOn: AssertEquals not returning expected value');
AssertEquals_BOOL(stStatusExpected.b1_ReadyForOperation, fbFSM.nStatus.b1_ReadyForOperation, 'b1_ReadyForOperation: AssertEquals not returning expected value');
AssertEquals_BOOL(stStatusExpected.b2_OperationEnabled, fbFSM.nStatus.b2_OperationEnabled, 'b2_OperationEnabled: AssertEquals not returning expected value');	
AssertEquals_BOOL(stStatusExpected.b6_SwitchingOnInhibited, fbFSM.nStatus.b6_SwitchingOnInhibited, 'b6_SwitchingOnInhibited: AssertEquals not returning expected value');	

TEST_FINISHED();
END_METHOD

METHOD TestState_S3 : BOOL
VAR
	fbFSM 				: FB_ProfidriveGSM;
	stStatusExpected	: ST_ProfidriveGSM_Status;
END_VAR
TEST('Set State S3');

//Arrange
fbFSM.eState := E_ProfidriveGSM_State.S3_SwitchedOn;

stStatusExpected.b0_ReadyToSwitchOn 		:= TRUE;				
stStatusExpected.b1_ReadyForOperation 		:= TRUE;				
stStatusExpected.b2_OperationEnabled 		:= FALSE;
stStatusExpected.b6_SwitchingOnInhibited 	:= FALSE;

//Act
fbFSM();

//Assert
AssertEquals_BOOL(stStatusExpected.b0_ReadyToSwitchOn, fbFSM.nStatus.b0_ReadyToSwitchOn, 'b0_ReadyToSwitchOn: AssertEquals not returning expected value');
AssertEquals_BOOL(stStatusExpected.b1_ReadyForOperation, fbFSM.nStatus.b1_ReadyForOperation, 'b1_ReadyForOperation: AssertEquals not returning expected value');
AssertEquals_BOOL(stStatusExpected.b2_OperationEnabled, fbFSM.nStatus.b2_OperationEnabled, 'b2_OperationEnabled: AssertEquals not returning expected value');	
AssertEquals_BOOL(stStatusExpected.b6_SwitchingOnInhibited, fbFSM.nStatus.b6_SwitchingOnInhibited, 'b6_SwitchingOnInhibited: AssertEquals not returning expected value');	

TEST_FINISHED();
END_METHOD

METHOD TestState_S4 : BOOL
VAR
	fbFSM 				: FB_ProfidriveGSM;
	stStatusExpected	: ST_ProfidriveGSM_Status;
END_VAR
TEST('Set State S4');

//Arrange
fbFSM.eState := E_ProfidriveGSM_State.S4_Operation;

stStatusExpected.b0_ReadyToSwitchOn 		:= TRUE;				
stStatusExpected.b1_ReadyForOperation 		:= TRUE;				
stStatusExpected.b2_OperationEnabled 		:= TRUE;
stStatusExpected.b6_SwitchingOnInhibited 	:= FALSE;

//Act
fbFSM();

//Assert
AssertEquals_BOOL(stStatusExpected.b0_ReadyToSwitchOn, fbFSM.nStatus.b0_ReadyToSwitchOn, 'b0_ReadyToSwitchOn: AssertEquals not returning expected value');
AssertEquals_BOOL(stStatusExpected.b1_ReadyForOperation, fbFSM.nStatus.b1_ReadyForOperation, 'b1_ReadyForOperation: AssertEquals not returning expected value');
AssertEquals_BOOL(stStatusExpected.b2_OperationEnabled, fbFSM.nStatus.b2_OperationEnabled, 'b2_OperationEnabled: AssertEquals not returning expected value');	
AssertEquals_BOOL(stStatusExpected.b6_SwitchingOnInhibited, fbFSM.nStatus.b6_SwitchingOnInhibited, 'b6_SwitchingOnInhibited: AssertEquals not returning expected value');	

TEST_FINISHED();
END_METHOD

METHOD TestState_S51 : BOOL
VAR
	fbFSM 				: FB_ProfidriveGSM;
	stStatusExpected	: ST_ProfidriveGSM_Status;
END_VAR
TEST('Set State S51');

//Arrange
fbFSM.eState := E_ProfidriveGSM_State.S51_RampStop;

stStatusExpected.b0_ReadyToSwitchOn 		:= TRUE;				
stStatusExpected.b1_ReadyForOperation 		:= TRUE;				
stStatusExpected.b2_OperationEnabled 		:= FALSE;
stStatusExpected.b6_SwitchingOnInhibited 	:= FALSE;

//Act
fbFSM();

//Assert
AssertEquals_BOOL(stStatusExpected.b0_ReadyToSwitchOn, fbFSM.nStatus.b0_ReadyToSwitchOn, 'b0_ReadyToSwitchOn: AssertEquals not returning expected value');
AssertEquals_BOOL(stStatusExpected.b1_ReadyForOperation, fbFSM.nStatus.b1_ReadyForOperation, 'b1_ReadyForOperation: AssertEquals not returning expected value');
AssertEquals_BOOL(stStatusExpected.b2_OperationEnabled, fbFSM.nStatus.b2_OperationEnabled, 'b2_OperationEnabled: AssertEquals not returning expected value');	
AssertEquals_BOOL(stStatusExpected.b6_SwitchingOnInhibited, fbFSM.nStatus.b6_SwitchingOnInhibited, 'b6_SwitchingOnInhibited: AssertEquals not returning expected value');	

TEST_FINISHED();
END_METHOD

METHOD TestState_S52 : BOOL
VAR
	fbFSM 				: FB_ProfidriveGSM;
	stStatusExpected	: ST_ProfidriveGSM_Status;
END_VAR
TEST('Set State S52');

//Arrange
fbFSM.eState := E_ProfidriveGSM_State.S52_QuickStop;

stStatusExpected.b0_ReadyToSwitchOn 		:= TRUE;				
stStatusExpected.b1_ReadyForOperation 		:= TRUE;				
stStatusExpected.b2_OperationEnabled 		:= FALSE;
stStatusExpected.b6_SwitchingOnInhibited 	:= FALSE;

//Act
fbFSM();

//Assert
AssertEquals_BOOL(stStatusExpected.b0_ReadyToSwitchOn, fbFSM.nStatus.b0_ReadyToSwitchOn, 'b0_ReadyToSwitchOn: AssertEquals not returning expected value');
AssertEquals_BOOL(stStatusExpected.b1_ReadyForOperation, fbFSM.nStatus.b1_ReadyForOperation, 'b1_ReadyForOperation: AssertEquals not returning expected value');
AssertEquals_BOOL(stStatusExpected.b2_OperationEnabled, fbFSM.nStatus.b2_OperationEnabled, 'b2_OperationEnabled: AssertEquals not returning expected value');	
AssertEquals_BOOL(stStatusExpected.b6_SwitchingOnInhibited, fbFSM.nStatus.b6_SwitchingOnInhibited, 'b6_SwitchingOnInhibited: AssertEquals not returning expected value');	

TEST_FINISHED();
END_METHOD

METHOD TestTransitions_S0 : BOOL
VAR
	fbFSM 				: FB_ProfidriveGSM;
	stStatusExpected	: ST_ProfidriveGSM_Status;
	nStatusExpected 	: WORD;
END_VAR
TEST('Transition S0>S0');

//Arrange
fbFSM.bPowerOn := FALSE;
fbFSM.eState := E_ProfidriveGSM_State.S0_Disabled;

//Act
fbFSM();

//Assert
AssertEquals_INT(E_ProfidriveGSM_State.S0_Disabled, fbFSM.eState, 'eState: AssertEquals not returning expected value');

TEST_FINISHED();


TEST('Transition S0>S1');

//Arrange
fbFSM.bPowerOn := TRUE;
fbFSM.eState := E_ProfidriveGSM_State.S0_Disabled;

//Act
fbFSM();

//Assert
AssertEquals_INT(E_ProfidriveGSM_State.S1_SwitchingOnInhibited, fbFSM.eState, 'eState: AssertEquals not returning expected value');

TEST_FINISHED();
END_METHOD

METHOD TestTransitions_S1 : BOOL
VAR
	fbFSM 				: FB_ProfidriveGSM;
	stStatusExpected	: ST_ProfidriveGSM_Status;
	nStatusExpected 	: WORD;
END_VAR
TEST('Transition S1>S2');

//Arrange
fbFSM.bPowerOn := TRUE;
fbFSM.eState := E_ProfidriveGSM_State.S1_SwitchingOnInhibited;

fbFSM.nControl.b0_On 				:= FALSE;
fbFSM.nControl.b1_CoastStop 		:= TRUE;
fbFSM.nControl.b2_QuickStop 		:= TRUE;

//Act
fbFSM();

//Assert
AssertEquals_INT(E_ProfidriveGSM_State.S2_ReadyForSwitchingOn, fbFSM.eState, 'eState: AssertEquals not returning expected value');

TEST_FINISHED();
END_METHOD

METHOD TestTransitions_S2 : BOOL
VAR
	fbFSM 				: FB_ProfidriveGSM;
	stStatusExpected	: ST_ProfidriveGSM_Status;
	nStatusExpected 	: WORD;
END_VAR
TEST('Transition S2>S1 Case_1');

//Arrange
fbFSM.bPowerOn := TRUE;
fbFSM.eState := E_ProfidriveGSM_State.S2_ReadyForSwitchingOn;

fbFSM.nControl.b0_On 				:= TRUE;
fbFSM.nControl.b1_CoastStop 		:= FALSE;
fbFSM.nControl.b2_QuickStop 		:= TRUE;

//Act
fbFSM();

//Assert
AssertEquals_INT(E_ProfidriveGSM_State.S1_SwitchingOnInhibited, fbFSM.eState, 'eState: AssertEquals not returning expected value');

TEST_FINISHED();


TEST('Transition S2>S1 Case_2');

//Arrange
fbFSM.bPowerOn := TRUE;
fbFSM.eState := E_ProfidriveGSM_State.S2_ReadyForSwitchingOn;

fbFSM.nControl.b0_On 				:= TRUE;
fbFSM.nControl.b1_CoastStop 		:= TRUE;
fbFSM.nControl.b2_QuickStop 		:= FALSE;

//Act
fbFSM();

//Assert
AssertEquals_INT(E_ProfidriveGSM_State.S1_SwitchingOnInhibited, fbFSM.eState, 'eState: AssertEquals not returning expected value');

TEST_FINISHED();


TEST('Transition S2 Still');

//Arrange
fbFSM.bPowerOn := TRUE;
fbFSM.eState := E_ProfidriveGSM_State.S2_ReadyForSwitchingOn;

fbFSM.nControl.b0_On 				:= FALSE;
fbFSM.nControl.b1_CoastStop 		:= TRUE;
fbFSM.nControl.b2_QuickStop 		:= TRUE;

//Act
fbFSM();

//Assert
AssertEquals_INT(E_ProfidriveGSM_State.S2_ReadyForSwitchingOn, fbFSM.eState, 'eState: AssertEquals not returning expected value');

TEST_FINISHED();


TEST('Transition S2>S3');

//Arrange
fbFSM.bPowerOn := TRUE;
fbFSM.eState := E_ProfidriveGSM_State.S2_ReadyForSwitchingOn;

fbFSM.nControl.b0_On 				:= TRUE;
fbFSM.nControl.b1_CoastStop 		:= TRUE;
fbFSM.nControl.b2_QuickStop 		:= TRUE;

//Act
fbFSM();

//Assert
AssertEquals_INT(E_ProfidriveGSM_State.S3_SwitchedOn, fbFSM.eState, 'eState: AssertEquals not returning expected value');

TEST_FINISHED();
END_METHOD

METHOD TestTransitions_S3 : BOOL
VAR
	fbFSM 				: FB_ProfidriveGSM;
	stStatusExpected	: ST_ProfidriveGSM_Status;
	nStatusExpected 	: WORD;
END_VAR
TEST('Transition S3>S1 Case_1');

//Arrange
fbFSM.bPowerOn := TRUE;
fbFSM.eState := E_ProfidriveGSM_State.S3_SwitchedOn;

fbFSM.nControl.b0_On 				:= TRUE;
fbFSM.nControl.b1_CoastStop 		:= FALSE;
fbFSM.nControl.b2_QuickStop 		:= TRUE;

//Act
fbFSM();

//Assert
AssertEquals_INT(E_ProfidriveGSM_State.S1_SwitchingOnInhibited, fbFSM.eState, 'eState: AssertEquals not returning expected value');

TEST_FINISHED();


TEST('Transition S3>S1 Case_2');

//Arrange
fbFSM.bPowerOn := TRUE;
fbFSM.eState := E_ProfidriveGSM_State.S3_SwitchedOn;

fbFSM.nControl.b0_On 				:= TRUE;
fbFSM.nControl.b1_CoastStop 		:= TRUE;
fbFSM.nControl.b2_QuickStop 		:= FALSE;

//Act
fbFSM();

//Assert
AssertEquals_INT(E_ProfidriveGSM_State.S1_SwitchingOnInhibited, fbFSM.eState, 'eState: AssertEquals not returning expected value');

TEST_FINISHED();


TEST('Transition S3 Still');

//Arrange
fbFSM.bPowerOn := TRUE;
fbFSM.eState := E_ProfidriveGSM_State.S3_SwitchedOn;

fbFSM.nControl.b0_On 				:= TRUE;
fbFSM.nControl.b1_CoastStop 		:= TRUE;
fbFSM.nControl.b2_QuickStop 		:= TRUE;
fbFSM.nControl.b3_EnableOperation  := FALSE;

//Act
fbFSM();

//Assert
AssertEquals_INT(E_ProfidriveGSM_State.S3_SwitchedOn, fbFSM.eState, 'eState: AssertEquals not returning expected value');

TEST_FINISHED();


TEST('Transition S3>S2');

//Arrange
fbFSM.bPowerOn := TRUE;
fbFSM.eState := E_ProfidriveGSM_State.S3_SwitchedOn;

fbFSM.nControl.b0_On 				:= FALSE;
fbFSM.nControl.b1_CoastStop 		:= TRUE;
fbFSM.nControl.b2_QuickStop 		:= TRUE;

//Act
fbFSM();

//Assert
AssertEquals_INT(E_ProfidriveGSM_State.S2_ReadyForSwitchingOn, fbFSM.eState, 'eState: AssertEquals not returning expected value');

TEST_FINISHED();


TEST('Transition S3>S4');

//Arrange
fbFSM.bPowerOn := TRUE;
fbFSM.eState := E_ProfidriveGSM_State.S3_SwitchedOn;

fbFSM.nControl.b0_On 				:= TRUE;
fbFSM.nControl.b1_CoastStop 		:= TRUE;
fbFSM.nControl.b2_QuickStop 		:= TRUE;
fbFSM.nControl.b3_EnableOperation  := TRUE;

//Act
fbFSM();

//Assert
AssertEquals_INT(E_ProfidriveGSM_State.S4_Operation, fbFSM.eState, 'eState: AssertEquals not returning expected value');

TEST_FINISHED();
END_METHOD

METHOD TestTransitions_S4 : BOOL
VAR
	fbFSM 				: FB_ProfidriveGSM;
	stStatusExpected	: ST_ProfidriveGSM_Status;
	nStatusExpected 	: WORD;
END_VAR
TEST('Transition S4>S1');

//Arrange
fbFSM.bPowerOn := TRUE;
fbFSM.eState := E_ProfidriveGSM_State.S4_Operation;

fbFSM.nControl.b0_On 				:= FALSE;
fbFSM.nControl.b1_CoastStop 		:= FALSE;
fbFSM.nControl.b2_QuickStop 		:= FALSE;

//Act
fbFSM();

//Assert
AssertEquals_INT(E_ProfidriveGSM_State.S1_SwitchingOnInhibited, fbFSM.eState, 'eState: AssertEquals not returning expected value');

TEST_FINISHED();


TEST('Transition S4>S52');

//Arrange
fbFSM.bPowerOn := TRUE;
fbFSM.eState := E_ProfidriveGSM_State.S4_Operation;

fbFSM.nControl.b0_On 				:= FALSE;
fbFSM.nControl.b1_CoastStop 		:= TRUE;
fbFSM.nControl.b2_QuickStop 		:= FALSE;

//Act
fbFSM();

//Assert
AssertEquals_INT(E_ProfidriveGSM_State.S52_QuickStop, fbFSM.eState, 'eState: AssertEquals not returning expected value');

TEST_FINISHED();


TEST('Transition S4>S51');

//Arrange
fbFSM.bPowerOn := TRUE;
fbFSM.eState := E_ProfidriveGSM_State.S4_Operation;

fbFSM.nControl.b0_On 				:= FALSE;
fbFSM.nControl.b1_CoastStop 		:= TRUE;
fbFSM.nControl.b2_QuickStop 		:= TRUE;
fbFSM.nControl.b3_EnableOperation 	:= FALSE;

//Act
fbFSM();

//Assert
AssertEquals_INT(E_ProfidriveGSM_State.S51_RampStop, fbFSM.eState, 'eState: AssertEquals not returning expected value');

TEST_FINISHED();


TEST('Transition S4>S3');

//Arrange
fbFSM.bPowerOn := TRUE;
fbFSM.eState := E_ProfidriveGSM_State.S4_Operation;

fbFSM.nControl.b0_On 				:= TRUE;
fbFSM.nControl.b1_CoastStop 		:= TRUE;
fbFSM.nControl.b2_QuickStop 		:= TRUE;
fbFSM.nControl.b3_EnableOperation 	:= FALSE;

//Act
fbFSM();

//Assert
AssertEquals_INT(E_ProfidriveGSM_State.S3_SwitchedOn, fbFSM.eState, 'eState: AssertEquals not returning expected value');

TEST_FINISHED();
END_METHOD

METHOD TestTransitions_S51 : BOOL
VAR
	fbFSM 				: FB_ProfidriveGSM;
	stStatusExpected	: ST_ProfidriveGSM_Status;
	nStatusExpected 	: WORD;
END_VAR
TEST('Transition S51 Still');

//Arrange
fbFSM.bPowerOn := TRUE;
fbFSM.eState := E_ProfidriveGSM_State.S51_RampStop;

fbFSM.bStandstill					:= FALSE;
fbFSM.nControl.b0_On 				:= FALSE;
fbFSM.nControl.b1_CoastStop 		:= TRUE;
fbFSM.nControl.b2_QuickStop 		:= TRUE;
fbFSM.nControl.b3_EnableOperation 	:= TRUE;

//Act
fbFSM();

//Assert
AssertEquals_INT(E_ProfidriveGSM_State.S51_RampStop, fbFSM.eState, 'eState: AssertEquals not returning expected value');

TEST_FINISHED();


TEST('Transition S51>S1');

//Arrange
fbFSM.bPowerOn := TRUE;
fbFSM.eState := E_ProfidriveGSM_State.S51_RampStop;

fbFSM.bStandstill					:= FALSE;
fbFSM.nControl.b0_On 				:= FALSE;
fbFSM.nControl.b1_CoastStop 		:= FALSE;
fbFSM.nControl.b2_QuickStop 		:= FALSE;
fbFSM.nControl.b3_EnableOperation 	:= FALSE;

//Act
fbFSM();

//Assert
AssertEquals_INT(E_ProfidriveGSM_State.S1_SwitchingOnInhibited, fbFSM.eState, 'eState: AssertEquals not returning expected value');

TEST_FINISHED();


TEST('Transition S51>S52');

//Arrange
fbFSM.bPowerOn := TRUE;
fbFSM.eState := E_ProfidriveGSM_State.S51_RampStop;

fbFSM.bStandstill					:= FALSE;
fbFSM.nControl.b0_On 				:= FALSE;
fbFSM.nControl.b1_CoastStop 		:= TRUE;
fbFSM.nControl.b2_QuickStop 		:= FALSE;
fbFSM.nControl.b3_EnableOperation 	:= TRUE;

//Act
fbFSM();

//Assert
AssertEquals_INT(E_ProfidriveGSM_State.S52_QuickStop, fbFSM.eState, 'eState: AssertEquals not returning expected value');

TEST_FINISHED();


TEST('Transition S51>S2 Case_1');

//Arrange
fbFSM.bPowerOn := TRUE;
fbFSM.eState := E_ProfidriveGSM_State.S51_RampStop;

fbFSM.bStandstill					:= FALSE;
fbFSM.nControl.b0_On 				:= FALSE;
fbFSM.nControl.b1_CoastStop 		:= TRUE;
fbFSM.nControl.b2_QuickStop 		:= TRUE;
fbFSM.nControl.b3_EnableOperation 	:= FALSE;

//Act
fbFSM();

//Assert
AssertEquals_INT(E_ProfidriveGSM_State.S2_ReadyForSwitchingOn, fbFSM.eState, 'eState: AssertEquals not returning expected value');

TEST_FINISHED();


TEST('Transition S51>S2 Case_2');

//Arrange
fbFSM.bPowerOn := TRUE;
fbFSM.eState := E_ProfidriveGSM_State.S51_RampStop;

fbFSM.bStandstill					:= TRUE;
fbFSM.nControl.b0_On 				:= FALSE;
fbFSM.nControl.b1_CoastStop 		:= TRUE;
fbFSM.nControl.b2_QuickStop 		:= TRUE;
fbFSM.nControl.b3_EnableOperation 	:= TRUE;

//Act
fbFSM();

//Assert
AssertEquals_INT(E_ProfidriveGSM_State.S2_ReadyForSwitchingOn, fbFSM.eState, 'eState: AssertEquals not returning expected value');

TEST_FINISHED();


TEST('Transition S51>S4');

//Arrange
fbFSM.bPowerOn := TRUE;
fbFSM.eState := E_ProfidriveGSM_State.S51_RampStop;

fbFSM.bStandstill					:= FALSE;
fbFSM.nControl.b0_On 				:= TRUE;
fbFSM.nControl.b1_CoastStop 		:= TRUE;
fbFSM.nControl.b2_QuickStop 		:= TRUE;
fbFSM.nControl.b3_EnableOperation 	:= TRUE;

//Act
fbFSM();

//Assert
AssertEquals_INT(E_ProfidriveGSM_State.S4_Operation, fbFSM.eState, 'eState: AssertEquals not returning expected value');

TEST_FINISHED();
END_METHOD

METHOD TestTransitions_S52 : BOOL
VAR
	fbFSM 				: FB_ProfidriveGSM;
	stStatusExpected	: ST_ProfidriveGSM_Status;
	nStatusExpected 	: WORD;
END_VAR
TEST('Transition S52 Still');

//Arrange
fbFSM.bPowerOn := TRUE;
fbFSM.eState := E_ProfidriveGSM_State.S52_QuickStop;

fbFSM.bStandstill					:= FALSE;
fbFSM.nControl.b0_On 				:= FALSE;
fbFSM.nControl.b1_CoastStop 		:= TRUE;
fbFSM.nControl.b2_QuickStop 		:= FALSE;
fbFSM.nControl.b3_EnableOperation 	:= TRUE;

//Act
fbFSM();

//Assert
AssertEquals_INT(E_ProfidriveGSM_State.S52_QuickStop, fbFSM.eState, 'eState: AssertEquals not returning expected value');

TEST_FINISHED();


TEST('Transition S51>S1 Case_1');

//Arrange
fbFSM.bPowerOn := TRUE;
fbFSM.eState := E_ProfidriveGSM_State.S52_QuickStop;

fbFSM.bStandstill					:= FALSE;
fbFSM.nControl.b0_On 				:= FALSE;
fbFSM.nControl.b1_CoastStop 		:= FALSE;
fbFSM.nControl.b2_QuickStop 		:= FALSE;
fbFSM.nControl.b3_EnableOperation 	:= FALSE;

//Act
fbFSM();

//Assert
AssertEquals_INT(E_ProfidriveGSM_State.S1_SwitchingOnInhibited, fbFSM.eState, 'eState: AssertEquals not returning expected value');

TEST_FINISHED();


TEST('Transition S52>S1 Case_2');

//Arrange
fbFSM.bPowerOn := TRUE;
fbFSM.eState := E_ProfidriveGSM_State.S52_QuickStop;

fbFSM.bStandstill					:= FALSE;
fbFSM.nControl.b0_On 				:= FALSE;
fbFSM.nControl.b1_CoastStop 		:= TRUE;
fbFSM.nControl.b2_QuickStop 		:= FALSE;
fbFSM.nControl.b3_EnableOperation 	:= FALSE;

//Act
fbFSM();

//Assert
AssertEquals_INT(E_ProfidriveGSM_State.S1_SwitchingOnInhibited, fbFSM.eState, 'eState: AssertEquals not returning expected value');

TEST_FINISHED();

TEST('Transition S52>S1 Case_3');

//Arrange
fbFSM.bPowerOn := TRUE;
fbFSM.eState := E_ProfidriveGSM_State.S52_QuickStop;

fbFSM.bStandstill					:= TRUE;
fbFSM.nControl.b0_On 				:= FALSE;
fbFSM.nControl.b1_CoastStop 		:= TRUE;
fbFSM.nControl.b2_QuickStop 		:= FALSE;
fbFSM.nControl.b3_EnableOperation 	:= TRUE;

//Act
fbFSM();

//Assert
AssertEquals_INT(E_ProfidriveGSM_State.S1_SwitchingOnInhibited, fbFSM.eState, 'eState: AssertEquals not returning expected value');

TEST_FINISHED();
END_METHOD

END_FUNCTION_BLOCK

// ---- Common/ProfidriveGSM/FB_ProfidriveGSM.TcPOU
// Profidrive General State Machine
FUNCTION_BLOCK PUBLIC FB_ProfidriveGSM
VAR_INPUT
	bPowerOn					: BOOL := TRUE;
	bStandstill					: BOOL;
	nControl					: ST_ProfidriveGSM_Control;
END_VAR

VAR_OUTPUT
	nStatus						: ST_ProfidriveGSM_Status;
END_VAR

VAR	
	_eState 					: E_ProfidriveGSM_State := E_ProfidriveGSM_State.S1_SwitchingOnInhibited;
END_VAR

CASE _eState OF 
	E_ProfidriveGSM_State.S0_Disabled : S0_Disabled();
	E_ProfidriveGSM_State.S1_SwitchingOnInhibited : S1_SwitchingOnInhibited();
	E_ProfidriveGSM_State.S2_ReadyForSwitchingOn : S2_ReadyForSwitchingOn();
	E_ProfidriveGSM_State.S3_SwitchedOn : S3_SwitchedOn();
	E_ProfidriveGSM_State.S4_Operation : S4_Operation();
	E_ProfidriveGSM_State.S51_RampStop : S51_RampStop();
	E_ProfidriveGSM_State.S52_QuickStop : S52_QuickStop();
END_CASE

PROPERTY eState : E_ProfidriveGSM_State
GET
eState := _eState;
END_GET
SET
_eState := eState;
END_SET
END_PROPERTY

{ attribute 'hide' }
METHOD PROTECTED S0_Disabled
nStatus.b0_ReadyToSwitchOn 			:= FALSE;				
nStatus.b1_ReadyForOperation 		:= FALSE;				
nStatus.b2_OperationEnabled 		:= FALSE;					
nStatus.b3_FaultPresent 			:= FALSE;						
nStatus.b4_CoastStop 				:= FALSE;	 					
nStatus.b5_QuickStop 				:= FALSE;						
nStatus.b6_SwitchingOnInhibited 	:= FALSE;				
nStatus.b7_WarningPresent			:= FALSE;			
nStatus.b9_ControlRequested 		:= FALSE;	

(*to S1*)	
IF bPowerOn THEN
	_eState := E_ProfidriveGSM_State.S1_SwitchingOnInhibited;
END_IF
END_METHOD

{ attribute 'hide' }
METHOD INTERNAL S1_SwitchingOnInhibited
VAR_INPUT
END_VAR
nStatus.b0_ReadyToSwitchOn 		:= FALSE;				
nStatus.b1_ReadyForOperation 		:= FALSE;				
nStatus.b2_OperationEnabled 		:= FALSE;						
nStatus.b6_SwitchingOnInhibited 	:= TRUE;

(*to S2_ReadyForSwitchingOn*)	
IF NOT nControl.b0_On AND nControl.b1_CoastStop AND nControl.b2_QuickStop THEN
	_eState := E_ProfidriveGSM_State.S2_ReadyForSwitchingOn;
END_IF
END_METHOD

{ attribute 'hide' }
METHOD INTERNAL S2_ReadyForSwitchingOn
VAR_INPUT
END_VAR
nStatus.b0_ReadyToSwitchOn 		:= TRUE;				
nStatus.b1_ReadyForOperation 		:= FALSE;				
nStatus.b2_OperationEnabled 		:= FALSE;						
nStatus.b6_SwitchingOnInhibited 	:= FALSE;

(*to S1_SwitchingOnInhibited*)	
IF NOT nControl.b1_CoastStop OR NOT nControl.b2_QuickStop THEN
	_eState := E_ProfidriveGSM_State.S1_SwitchingOnInhibited;
	RETURN;
END_IF

(*to S3_SwitchedOn*)	
IF nControl.b0_On THEN
	_eState := E_ProfidriveGSM_State.S3_SwitchedOn;
END_IF
END_METHOD

{ attribute 'hide' }
METHOD INTERNAL S3_SwitchedOn
VAR_INPUT
END_VAR
nStatus.b0_ReadyToSwitchOn 		:= TRUE;				
nStatus.b1_ReadyForOperation 		:= TRUE;				
nStatus.b2_OperationEnabled 		:= FALSE;						
nStatus.b6_SwitchingOnInhibited 	:= FALSE;

(*to S1_SwitchingOnInhibited*)	
IF NOT nControl.b1_CoastStop OR NOT nControl.b2_QuickStop THEN
	_eState := E_ProfidriveGSM_State.S1_SwitchingOnInhibited;
	RETURN;
END_IF

(*to S2_ReadyForSwitchingOn*)	
IF NOT nControl.b0_On THEN
	_eState := E_ProfidriveGSM_State.S2_ReadyForSwitchingOn;
	RETURN;
END_IF

(*to S4_Operation*)	
IF nControl.b3_EnableOperation THEN
	_eState := E_ProfidriveGSM_State.S4_Operation;
END_IF
END_METHOD

{ attribute 'hide' }
METHOD INTERNAL S4_Operation
VAR_INPUT
END_VAR
nStatus.b0_ReadyToSwitchOn 		:= TRUE;				
nStatus.b1_ReadyForOperation 		:= TRUE;				
nStatus.b2_OperationEnabled 		:= TRUE;					
nStatus.b6_SwitchingOnInhibited 	:= FALSE;

(*to S1_SwitchingOnInhibited*)	
IF NOT nControl.b1_CoastStop THEN
	_eState := E_ProfidriveGSM_State.S1_SwitchingOnInhibited;
	RETURN;
END_IF

(*to S52_QuickStop*)	
IF NOT nControl.b2_QuickStop THEN
	_eState := E_ProfidriveGSM_State.S52_QuickStop;
	RETURN;
END_IF

(*to S51_RampStop*)	
IF NOT nControl.b0_On THEN
	_eState := E_ProfidriveGSM_State.S51_RampStop;
	RETURN;
END_IF

(*to S3_SwitchedOn*)	
IF NOT nControl.b3_EnableOperation THEN
	_eState := E_ProfidriveGSM_State.S3_SwitchedOn;
END_IF
END_METHOD

{ attribute 'hide' }
METHOD INTERNAL S51_RampStop
VAR_INPUT
END_VAR
nStatus.b0_ReadyToSwitchOn 		:= TRUE;				
nStatus.b1_ReadyForOperation 		:= TRUE;				
nStatus.b2_OperationEnabled 		:= FALSE;					
nStatus.b6_SwitchingOnInhibited 	:= FALSE;

(*to S1_SwitchingOnInhibited*)	
IF NOT nControl.b1_CoastStop THEN
	_eState := E_ProfidriveGSM_State.S1_SwitchingOnInhibited;
	RETURN;
END_IF

(*to S52_QuickStop*)	
IF NOT nControl.b2_QuickStop THEN
	_eState := E_ProfidriveGSM_State.S52_QuickStop;
	RETURN;
END_IF

(*to S2_ReadyForSwitchingOn*)	
IF NOT nControl.b3_EnableOperation OR bStandstill THEN
	_eState := E_ProfidriveGSM_State.S2_ReadyForSwitchingOn;
END_IF

(*to S4_Operation*)	
IF nControl.b0_On THEN
	_eState := E_ProfidriveGSM_State.S4_Operation;
	RETURN;
END_IF
END_METHOD

{ attribute 'hide' }
METHOD INTERNAL S52_QuickStop
VAR_INPUT
END_VAR
nStatus.b0_ReadyToSwitchOn 		:= TRUE;				
nStatus.b1_ReadyForOperation 	:= TRUE;				
nStatus.b2_OperationEnabled 	:= FALSE;					
nStatus.b6_SwitchingOnInhibited := FALSE;

(*to S1_SwitchingOnInhibited*)	
IF NOT nControl.b1_CoastStop THEN
	_eState := E_ProfidriveGSM_State.S1_SwitchingOnInhibited;
	RETURN;
END_IF

(*to S1_SwitchingOnInhibited*)	
IF NOT nControl.b3_EnableOperation OR bStandstill THEN
	_eState := E_ProfidriveGSM_State.S1_SwitchingOnInhibited;
END_IF
END_METHOD

END_FUNCTION_BLOCK

// ---- Tests/Devices/FB_ProfidriveTelegram1_Test.TcPOU
FUNCTION_BLOCK FB_ProfidriveTelegram1_Test EXTENDS TcUnit.FB_TestSuite

Test_ProcessDataControl();
Test_ProcessDataStatus();
Test_Cycle_Status_Const_Mirror();

METHOD Test_Cycle_Status_Const_Mirror : REFERENCE TO FB_Test
VAR
	fbDrive 			: FB_Profidrive_Telegram1;
	bExpected			: BOOL;
	stExpected			: ST_Profidrive_Telegram1_Status;
	bResult 			: BOOL;	
	stResult			: ST_Profidrive_Telegram1_Status;
	
	stSetControl		: ST_Profidrive_Telegram1_Control;
END_VAR
TEST('Status CONST TRUE');

bExpected := TRUE;

fbDrive.Cycle();

stResult := fbDrive.stStatus;

bResult := BIT_TO_BOOL(stResult.b8_DeviationWithinTolerance);

AssertEquals(Expected := bExpected,
             Actual := bResult,
             Message := 'DeviationWithinTolerance not set correctly');

bResult := BIT_TO_BOOL(stResult.b11_TorqueOrPowerLimitNotReached);
			 
AssertEquals(Expected := bExpected,
             Actual := bResult,
             Message := 'TorqueOrPowerLimitNotReached not set correctly');
			 
bResult := BIT_TO_BOOL(stResult.b13_NoOvertempAlarm);
			 
AssertEquals(Expected := bExpected,
             Actual := bResult,
             Message := 'NoOvertempAlarm not set correctly');

bResult := BIT_TO_BOOL(stResult.b15_NoAlarmNoOvertempPowerUnit);
			 
AssertEquals(Expected := bExpected,
             Actual := bResult,
             Message := 'NoAlarmNoOvertempPowerUnit not set correctly');
	 
TEST_FINISHED();

TEST('Status CONST FALSE');

bExpected := FALSE;

fbDrive.Cycle();

stResult := fbDrive.stStatus;

bResult := BIT_TO_BOOL(stResult.b3_FaultPresent);

AssertEquals(Expected := bExpected,
             Actual := bResult,
             Message := 'FaultPresent not set correctly');

bResult := BIT_TO_BOOL(stResult.b7_AlarmPresent);
			 
AssertEquals(Expected := bExpected,
             Actual := bResult,
             Message := 'AlarmPresent not set correctly');
TEST_FINISHED();

TEST('Status Mirror Control FALSE');

bExpected := FALSE;

stSetControl.b3_EnableOperation := bExpected;

fbDrive.stConfig.bControlRequested := bExpected;

fbDrive.stControl := stSetControl;

fbDrive.Cycle();

stResult := fbDrive.stStatus;

bResult := BIT_TO_BOOL(stResult.b2_OperationEnabled);
			 
AssertEquals(Expected := bExpected,
             Actual := bResult,
             Message := 'OperationEnabled not set correctly');

bResult := BIT_TO_BOOL(stResult.b9_ControlRequested);
			 
AssertEquals(Expected := bExpected,
             Actual := bResult,
             Message := 'ControlRequested not set correctly');

TEST_FINISHED();

TEST('Status Mirror Control TRUE');

bExpected := TRUE;

stSetControl.b3_EnableOperation := bExpected;

fbDrive.stConfig.bControlRequested := bExpected;

fbDrive.stControl := stSetControl;

fbDrive.Cycle();

stResult := fbDrive.stStatus;

bResult := BIT_TO_BOOL(stResult.b2_OperationEnabled);
			 
AssertEquals(Expected := bExpected,
             Actual := bResult,
             Message := 'OperationEnabled not set correctly');

bResult := BIT_TO_BOOL(stResult.b9_ControlRequested);
			 
AssertEquals(Expected := bExpected,
             Actual := bResult,
             Message := 'ControlRequested not set correctly');
	 
TEST_FINISHED();
END_METHOD

METHOD Test_ProcessDataControl : REFERENCE TO FB_Test
VAR
	fbDrive 					: FB_Profidrive_Telegram1;
	
	nExpectedSTW1 				: WORD;
	nExpectedTargetVelocity 	: INT;
	nActualSTW1 				: WORD;
	nActualTargetVelocity		: INT;	
		
	aExpectedControlData 		: ST_Profidrive_Telegram1_Control;		
	aActualControlData			: ST_Profidrive_Telegram1_Control;	
END_VAR
TEST('Process data to control structure');

//Arrange
nExpectedSTW1 := 16#A1B2;
nExpectedTargetVelocity := UINT_TO_INT(16#C3D4);

F_Memcpy(ADR(aExpectedControlData), ADR(nExpectedSTW1), 2, FALSE);
F_Memcpy(ADR(aExpectedControlData) + 2, ADR(nExpectedTargetVelocity), 2, FALSE);

fbDrive.pControl := ADR(aExpectedControlData);

//Act
fbDrive.GetControlData();

//Assert
F_Memcpy(ADR(nActualSTW1), ADR(fbDrive.stControl), 2, FALSE);
F_Memcpy(ADR(nActualTargetVelocity), ADR(fbDrive.stControl) + 2, 2, FALSE);

AssertEquals(Expected := nExpectedSTW1,
             Actual := nActualSTW1,
             Message := 'STW1 is not correct');
	 
AssertEquals(Expected := nExpectedTargetVelocity,
             Actual := nActualTargetVelocity,
             Message := 'TargetVelocity is not correct');

TEST_FINISHED();


TEST('Process data to control structure SWAP');

//Arrange
nExpectedSTW1 := 16#C3F3;
nExpectedTargetVelocity := UINT_TO_INT(16#C3F3);

F_Memcpy(ADR(aExpectedControlData), ADR(nExpectedSTW1), 2, TRUE);
F_Memcpy(ADR(aExpectedControlData) + 2, ADR(nExpectedTargetVelocity), 2, TRUE);

fbDrive.stConfig.bSwapProcessData := TRUE;

fbDrive.pControl := ADR(aExpectedControlData);

//Act
fbDrive.GetControlData();

//Assert
F_Memcpy(ADR(nActualSTW1), ADR(fbDrive.stControl), 2, FALSE);
F_Memcpy(ADR(nActualTargetVelocity), ADR(fbDrive.stControl) + 2, 2, FALSE);

AssertEquals(Expected := nExpectedSTW1,
             Actual := nActualSTW1,
             Message := 'STW1 is not correct');
	 
AssertEquals(Expected := nExpectedTargetVelocity,
             Actual := nActualTargetVelocity,
             Message := 'TargetVelocity is not correct');	

TEST_FINISHED();
END_METHOD

METHOD Test_ProcessDataStatus : REFERENCE TO FB_Test
VAR
	fbDrive 					: FB_Profidrive_Telegram1;
	
	nExpectedZSW1 				: WORD;
	nExpectedActualVelocity		: INT;	
	nActualZSW1 				: WORD;
	nActualActualVelocity		: INT;	

	stExpectedStatusData 		: ST_Profidrive_Telegram1_Status;		
	stActualStatusData 			: ST_Profidrive_Telegram1_Status;	
END_VAR
TEST('Assign status structure to process data');

//Arrange
nExpectedZSW1 := 16#A1B2;
nExpectedActualVelocity := UINT_TO_INT(16#C3D4);
F_Memcpy(ADR(fbDrive.stStatus), ADR(nExpectedZSW1), 2, FALSE);
F_Memcpy(ADR(fbDrive.stStatus) + 2, ADR(nExpectedActualVelocity), 2, FALSE);

fbDrive.pStatus := ADR(stActualStatusData);

//Act
fbDrive.SetStatusData();

//Assert
F_Memcpy(ADR(nActualZSW1), ADR(stActualStatusData), 2, FALSE);
F_Memcpy(ADR(nActualActualVelocity), ADR(stActualStatusData) + 2, 2, FALSE);

AssertEquals(Expected := nExpectedZSW1,
             Actual := nActualZSW1,
             Message := 'ZSW1 is not correct');
	 
AssertEquals(Expected := nExpectedActualVelocity,
             Actual := nActualActualVelocity,
             Message := 'ActualVelocity is not correct');	

TEST_FINISHED();


TEST('Assign status structure to process data SWAP');

//Arrange
nExpectedZSW1 := 16#A1B2;
nExpectedActualVelocity	:= UINT_TO_INT(16#C3D4);

F_Memcpy(ADR(fbDrive.stStatus), ADR(nExpectedZSW1), 2, FALSE);
F_Memcpy(ADR(fbDrive.stStatus) + 2, ADR(nExpectedActualVelocity), 2, FALSE);

fbDrive.stConfig.bSwapProcessData := TRUE;
fbDrive.pStatus := ADR(stActualStatusData);

//Act
fbDrive.SetStatusData();

//Assert
F_Memcpy(ADR(nActualZSW1), ADR(stActualStatusData), 2, TRUE);
F_Memcpy(ADR(nActualActualVelocity), ADR(stActualStatusData) + 2, 2, TRUE);

AssertEquals(Expected := nExpectedZSW1,
             Actual := nActualZSW1,
             Message := 'ZSW1 is not correct');
	 
AssertEquals(Expected := nExpectedActualVelocity,
             Actual := nActualActualVelocity,
             Message := 'ActualVelocity is not correct');	

TEST_FINISHED();
END_METHOD

END_FUNCTION_BLOCK

// ---- Devices/Profidrive_Telegram1/FB_Profidrive_Telegram1.TcPOU
{attribute 'reflection'} 
FUNCTION_BLOCK FB_Profidrive_Telegram1 EXTENDS FB_LinkDataReal
VAR_INPUT	
	pControl 			: PVOID; //Pocess data from fieldbus. Size must be >= stControl.
	pStatus 			: PVOID; //Pocess data to fieldbus. Size must be >= stStatus.
	stControl 			: ST_Profidrive_Telegram1_Control; //Control structure. Is read from the fieldbus.
	stConfig 			: ST_Profidrive_Telegram1_Config; //Config structure. Contains parameters of the device.	
END_VAR

VAR_OUTPUT
	stStatus					: ST_Profidrive_Telegram1_Status;
	fValue						: REAL;
END_VAR

VAR
    {attribute 'instance-path'} 
    {attribute 'noinit'} 
    _sPath 						: STRING; 	
	                        	
	_fbProfidriveGSM			: FB_ProfidriveGSM;	
	_fbMoveVelocity				: FB_MoveVelocity;
	                        	
	_fAcceleration	 			: REAL;
	_fDeceleration		 		: REAL;
	_fDecelerationQuickStop 	: REAL;
	_fDecelerationCoastStop 	: REAL;
	_bQuickStopExternal			: BOOL;	
END_VAR

SUPER^();
InitRun();

GetControlData();
Cycle();
SetStatusData();

METHOD INTERNAL Cycle
(*Initialize Init Value*)
IF SUPER^.Status.7 THEN
	ControlData := StatusData;
END_IF

(* Call base statemachine *)
_fbProfidriveGSM.bStandstill					:= OC_Core.F_Compare(_fbMoveVelocity.fVelocity, 0, 1E-3);
_fbProfidriveGSM.nControl.b0_On 				:= stControl.b0_OFF1;
_fbProfidriveGSM.nControl.b1_CoastStop 			:= stControl.b1_OFF2;
_fbProfidriveGSM.nControl.b2_QuickStop 			:= stControl.b2_OFF3 AND NOT _bQuickStopExternal;
_fbProfidriveGSM.nControl.b3_EnableOperation	:= stControl.b3_EnableOperation;

(* Preset target values *)
_fbMoveVelocity.fTargetVelocity					:= 0;
_fbMoveVelocity.fAccMax 						:= _fAcceleration;
_fbMoveVelocity.fDecMax 						:= _fDeceleration;

(* Operation Logic *)
Operation();
	
(* Coast stop, Quick stop, Ramp stop *)
IF _fbProfidriveGSM.eState = E_ProfidriveGSM_State.S1_SwitchingOnInhibited THEN
	_fbMoveVelocity.fTargetVelocity := 0;
	_fbMoveVelocity.fAccMax := _fDecelerationCoastStop;
	_fbMoveVelocity.fDecMax := _fDecelerationCoastStop;
ELSIF _fbProfidriveGSM.eState = E_ProfidriveGSM_State.S52_QuickStop THEN
	_fbMoveVelocity.fTargetVelocity := 0;
	_fbMoveVelocity.fAccMax := _fDecelerationQuickStop;
	_fbMoveVelocity.fDecMax := _fDecelerationQuickStop;
ELSIF _fbProfidriveGSM.eState = E_ProfidriveGSM_State.S51_RampStop THEN
	_fbMoveVelocity.fTargetVelocity := 0;
	_fbMoveVelocity.fAccMax := _fDeceleration;
	_fbMoveVelocity.fDecMax := _fDeceleration;
END_IF

(* Call MoveVelocity *)
_fbMoveVelocity();
	
(* Status word *)
stStatus.b0_ReadyForSwitchingOn				:= _fbProfidriveGSM.nStatus.b0_ReadyToSwitchOn;	
stStatus.b1_ReadyForOperation				:= _fbProfidriveGSM.nStatus.b1_ReadyForOperation;
stStatus.b2_OperationEnabled				:= stControl.b3_EnableOperation;
stStatus.b3_FaultPresent					:= FALSE;
stStatus.b4_NoCoastDownActive				:= _fbProfidriveGSM.eState <> E_ProfidriveGSM_State.S1_SwitchingOnInhibited;
stStatus.b5_NoQuickStopActive				:= _fbProfidriveGSM.eState <> E_ProfidriveGSM_State.S52_QuickStop;
stStatus.b6_SwitchingOnInhibited			:= _fbProfidriveGSM.nStatus.b6_SwitchingOnInhibited;
stStatus.b7_AlarmPresent					:= FALSE;
stStatus.b8_DeviationWithinTolerance		:= TRUE;
stStatus.b9_ControlRequested				:= stConfig.bControlRequested;
stStatus.b10_RpmCompValueReachedOrExceeded	:= _fbMoveVelocity.bIsReached;
stStatus.b11_TorqueOrPowerLimitNotReached	:= TRUE;
stStatus.b12_OpenHoldingBrake 				:= _fbProfidriveGSM.eState > E_ProfidriveGSM_State.S3_SwitchedOn;
stStatus.b13_NoOvertempAlarm				:= TRUE;	
stStatus.b14_MotorRotatesForwards			:= _fbMoveVelocity.fVelocity >= 0;
stStatus.b15_NoAlarmNoOvertempPowerUnit		:= TRUE;

(* Reset quickstop from extern *)
IF stControl.b7_AcknowledgeFaults THEN
	_bQuickStopExternal := FALSE;
END_IF

(* Calculate NIST *)
IF stConfig.fP2000 = 0 THEN
	stStatus.nVelocity	:= 0;
ELSE
	stStatus.nVelocity := REAL_TO_INT((_fbMoveVelocity.fVelocity * 16#4000) / stConfig.fP2000);
END_IF

(* Output of actual value *)	
IF stConfig.bOutputVelocity THEN
	ControlData := _fbMoveVelocity.fVelocity;
ELSE
	ControlData := ControlData + _fbMoveVelocity.fVelocity *  GVL_Core.fbSystem.fDeltaTime * GVL_Core.fbSystem.fTimeScaling;
END_IF

fValue := ControlData;
END_METHOD

METHOD INTERNAL GetControlData : BOOL
IF pControl <= 0 OR stConfig.bForceMode THEN RETURN; END_IF

F_Memcpy(ADR(stControl), pControl, 2, stConfig.bSwapProcessData);
F_Memcpy(ADR(stControl) + 2, pControl + 2, 2, stConfig.bSwapProcessData);
END_METHOD

METHOD INTERNAL InitRun : BOOL
VAR_INST
	bInitRun : BOOL := TRUE;
END_VAR
IF NOT bInitRun THEN RETURN; END_IF
bInitRun := FALSE;

IF pControl = 0 OR pStatus = 0 THEN
	ADSLOGSTR(ADSLOG_MSGTYPE_WARN, CONCAT(_sPath, ': %s'), 'Plc address not set.');
END_IF
END_METHOD

METHOD PRIVATE Operation : BOOL
IF _fbProfidriveGSM.eState = E_ProfidriveGSM_State.S4_Operation THEN	
	// Main setpoint
	IF NOT stControl.b8_Jog1 AND NOT stControl.b9_Jog2 THEN
		_fbMoveVelocity.fTargetVelocity := (stControl.nTargetVelocity * stConfig.fP2000) / 16#4000;
	// Jog 1
	ELSIF stControl.b8_Jog1 AND NOT stControl.b9_Jog2 THEN
		_fbMoveVelocity.fTargetVelocity := stConfig.fP1058;
	// Jog 2
	ELSIF NOT stControl.b8_Jog1 AND stControl.b9_Jog2 THEN	
		_fbMoveVelocity.fTargetVelocity := stConfig.fP1059;
	END_IF
	// Stop
	IF NOT stControl.b4_OperatingCondition OR NOT stControl.b6_EnableSetpoint THEN
		_fbMoveVelocity.fTargetVelocity := 0;
	END_IF
	// Invert velocity
	IF stControl.b11_SetpointInversion THEN
		_fbMoveVelocity.fTargetVelocity := -_fbMoveVelocity.fTargetVelocity;
	END_IF	
	// Hold velocity
	IF NOT stControl.b5_ContinueRampFunctionGenerator AND NOT stControl.b8_Jog1 AND NOT stControl.b9_Jog2 THEN
		_fbMoveVelocity.fTargetVelocity := _fbMoveVelocity.fVelocity;
	END_IF	
END_IF
END_METHOD

METHOD INTERNAL SetStatusData
IF pStatus <= 0 THEN RETURN; END_IF

F_Memcpy(pStatus, ADR(stStatus), 2, stConfig.bSwapProcessData);
F_Memcpy(pStatus + 2, ADR(stStatus) + 2, 2, stConfig.bSwapProcessData);
END_METHOD

END_FUNCTION_BLOCK

// ---- Tests/Devices/FB_SEW_MoviC_Position_Test.TcPOU
FUNCTION_BLOCK FB_SEW_MoviC_Position_Test EXTENDS TcUnit.FB_TestSuite

Test_ProcessDataControl();
Test_ProcessDataStatus();
Test_Safety();
Test_Cycle_Status_Const_Mirror();

Test_Cycle_Status_OperationMode('Test Target Mode EnergyOptimized',E_SEW_MoviC_Position_OperationMode.EnergyOptimized);
Test_Cycle_Status_OperationMode('Test Target Mode Jog',E_SEW_MoviC_Position_OperationMode.Jog);
Test_Cycle_Status_OperationMode('Test Target Mode JogNoEnc',E_SEW_MoviC_Position_OperationMode.JogNoEnc);
Test_Cycle_Status_OperationMode('Test Target Mode MechanicsOptimized',E_SEW_MoviC_Position_OperationMode.MechanicsOptimized);
Test_Cycle_Status_OperationMode('Test Target Mode PositionAbs',E_SEW_MoviC_Position_OperationMode.PositionAbs);
Test_Cycle_Status_OperationMode('Test Target Mode PositionModNeg',E_SEW_MoviC_Position_OperationMode.PositionModNeg);
Test_Cycle_Status_OperationMode('Test Target Mode PositionModPos',E_SEW_MoviC_Position_OperationMode.PositionModPos);
Test_Cycle_Status_OperationMode('Test Target Mode PositionModShort',E_SEW_MoviC_Position_OperationMode.PositionModShort);
Test_Cycle_Status_OperationMode('Test Target Mode PositionRel',E_SEW_MoviC_Position_OperationMode.PositionRel);
Test_Cycle_Status_OperationMode('Test Target Mode ReferenceBus',E_SEW_MoviC_Position_OperationMode.ReferenceBus);
Test_Cycle_Status_OperationMode('Test Target Mode ReferenceParam',E_SEW_MoviC_Position_OperationMode.ReferenceParam);
Test_Cycle_Status_OperationMode('Test Target Mode SpeedControl',E_SEW_MoviC_Position_OperationMode.SpeedControl);


Test_Cycle_Status_BrakeReleased('Test BrakeReleased; b1_EnableBusStop FALSE, b3_ReleaseBrake FALSE',FALSE,FALSE,FALSE);
Test_Cycle_Status_BrakeReleased('Test BrakeReleased; b1_EnableBusStop TRUE, b3_ReleaseBrake FALSE',TRUE,FALSE,TRUE);
Test_Cycle_Status_BrakeReleased('Test BrakeReleased; b1_EnableBusStop FALSE, b3_ReleaseBrake TRUE',FALSE,TRUE,TRUE);
Test_Cycle_Status_BrakeReleased('Test BrakeReleased; b1_EnableBusStop TRUE, b3_ReleaseBrake TRUE',TRUE,TRUE,TRUE);

Test_Cycle_Softwarelimits('Test Without Softwarelimi post',TRUE,-1000,1000, 2000, 2000);
Test_Cycle_Softwarelimits('Test Without Softwarelimit neg',TRUE,-1000,1000, -2000, -2000);

Test_Cycle_Softwarelimits('Test Softwarelimi post',FALSE,-1000,1000, 2000, 1000);
Test_Cycle_Softwarelimits('Test Softwarelimit neg',FALSE,-1000,1000, -2000, -1000);

METHOD Test_Cycle_Softwarelimits : REFERENCE TO FB_Test
VAR_INPUT
	sName 					: T_MaxString;
	bDisableSoftwareLimits 	: BOOL;
	nSoftwareLimitMin 		: DINT;
	nSoftwareLimitMax 		: DINT;
	nSetPosition			: DINT;
	nExpectedPosition		: DINT;
END_VAR
VAR
	fbDrive 			: FB_SEW_MoviC_Position;
	nResult 			: DINT;	
	nCycle				: UDINT;
	bIsPositionReached: INT;
END_VAR
TEST(sName);

fbDrive.stControl.b12_DisableSoftwareLimits := bDisableSoftwareLimits;
fbDrive.stConfig.nSoftwareLimitMin := nSoftwareLimitMin;
fbDrive.stConfig.nSoftwareLimitMax := nSoftwareLimitMax;

fbDrive.stControl.nSetpointSpeed := 32767;
fbDrive.stControl.nSetpointAcceleration := 32767;
fbDrive.stControl.nSetpointDeceleration := 32767;

fbDrive.stControl.nTargetApplicationMode := E_SEW_MoviC_Position_OperationMode.PositionAbs;
fbDrive.bSTO := TRUE;
fbDrive.stControl.b1_EnableBusStop := TRUE;
fbDrive.stControl.b13_ActivateInhibit := FALSE;
fbDrive.stControl.b0_EnableEStop := TRUE;
fbDrive.stControl.b7_StartStop := TRUE;

fbDrive.stControl.nTargetPosition := nSetPosition;

FOR nCycle := 1 TO 10000 DO
	fbDrive.Cycle();
END_FOR

nResult := fbDrive.stStatus.nActualPosition;

AssertEquals(Expected := nExpectedPosition,
             Actual := nResult,
             Message := 'Softwarelimits not used correctly');
	 
TEST_FINISHED();
END_METHOD

METHOD Test_Cycle_Status_BrakeReleased : REFERENCE TO FB_Test
VAR_INPUT
	sName 				: T_MaxString;
	b1_EnableBusStop 	: BOOL;
	b3_ReleaseBrake 	: BOOL;
	bExpected 			: BOOL;
END_VAR
VAR
	fbDrive 			: FB_SEW_MoviC_Position;
	bResult 			: BOOL;	
END_VAR
TEST(sName);

fbDrive.stControl.b1_EnableBusStop := b1_EnableBusStop;
fbDrive.stControl.b3_ReleaseBrake := b3_ReleaseBrake;

fbDrive.Cycle();

bResult := fbDrive.stStatus.b3_BrakeReleased;

AssertEquals(Expected := bExpected,
             Actual := bResult,
             Message := 'BrakeReleased not set correctly');
	 
TEST_FINISHED();
END_METHOD

METHOD Test_Cycle_Status_Const_Mirror : REFERENCE TO FB_Test
VAR
	fbDrive 			: FB_SEW_MoviC_Position;
	bExpected			: BOOL;
	stExpected			: ST_SEW_MoviC_Position_Status;
	bResult 			: BOOL;	
	stResult			: ST_SEW_MoviC_Position_Status;
	
	stSetControl		: ST_SEW_MoviC_Position_Control;
END_VAR
TEST('Status CONST TRUE');

bExpected := TRUE;

fbDrive.Cycle();

stResult := fbDrive.stStatus;

bResult := BIT_TO_BOOL(stResult.b0_InverterReady);

AssertEquals(Expected := bExpected,
             Actual := bResult,
             Message := 'InverterReady not set correctly');

bResult := BIT_TO_BOOL(stResult.b5_DriveReferenced);
			 
AssertEquals(Expected := bExpected,
             Actual := bResult,
             Message := 'DriveReferenced not set correctly');
	 
TEST_FINISHED();

TEST('Status CONST FALSE');

bExpected := FALSE;

fbDrive.Cycle();

stResult := fbDrive.stStatus;

bResult := BIT_TO_BOOL(stResult.b6_SetpointsActive);

AssertEquals(Expected := bExpected,
             Actual := bResult,
             Message := 'SetpointsActive not set correctly');

bResult := BIT_TO_BOOL(stResult.b8_ErrorActive);
			 
AssertEquals(Expected := bExpected,
             Actual := bResult,
             Message := 'ErrorActive not set correctly');

bResult := BIT_TO_BOOL(stResult.b9_WarningActive);
			 
AssertEquals(Expected := bExpected,
             Actual := bResult,
             Message := 'WarningActive not set correctly');
	 
TEST_FINISHED();

TEST('Status Mirror Control FALSE');

bExpected := FALSE;

stSetControl.b13_ActivateInhibit := bExpected;
stSetControl.b10_ActivateDriveTrain2 := bExpected;
stSetControl.b12_DisableSoftwareLimits := bExpected;
stSetControl.b14_ActivateStandByMode := bExpected;
stSetControl.b15_MovikitHeartbeat := bExpected;

fbDrive.stControl := stSetControl;

fbDrive.Cycle();

stResult := fbDrive.stStatus;

bResult := BIT_TO_BOOL(stResult.b10_DriveTrain2Active);
			 
AssertEquals(Expected := bExpected,
             Actual := bResult,
             Message := 'riveTrain2Active not set correctly');

bResult := BIT_TO_BOOL(stResult.b12_SoftwareLimitsDisabled);
			 
AssertEquals(Expected := bExpected,
             Actual := bResult,
             Message := 'SoftwareLimitsDisabled not set correctly');
			 
 bResult := BIT_TO_BOOL(stResult.b14_StandByModeActive);
			 
AssertEquals(Expected := bExpected,
             Actual := bResult,
             Message := 'StandByModeActive not set correctly');
			 
bResult := BIT_TO_BOOL(stResult.b15_MovikitHeartbeat);
			 
AssertEquals(Expected := bExpected,
             Actual := bResult,
             Message := 'MovikitHeartbeat not set correctly');
	 
TEST_FINISHED();

TEST('Status Mirror Control TRUE');

bExpected := TRUE;

stSetControl.b13_ActivateInhibit := bExpected;
stSetControl.b10_ActivateDriveTrain2 := bExpected;
stSetControl.b12_DisableSoftwareLimits := bExpected;
stSetControl.b14_ActivateStandByMode := bExpected;
stSetControl.b15_MovikitHeartbeat := bExpected;

fbDrive.stControl := stSetControl;

fbDrive.Cycle();

stResult := fbDrive.stStatus;

bResult := BIT_TO_BOOL(stResult.b2_PowerStageOn);

AssertEquals(Expected := bExpected,
             Actual := bResult,
             Message := 'PowerStageOn not set correctly');

bResult := BIT_TO_BOOL(stResult.b10_DriveTrain2Active);
			 
AssertEquals(Expected := bExpected,
             Actual := bResult,
             Message := 'riveTrain2Active not set correctly');

bResult := BIT_TO_BOOL(stResult.b12_SoftwareLimitsDisabled);
			 
AssertEquals(Expected := bExpected,
             Actual := bResult,
             Message := 'SoftwareLimitsDisabled not set correctly');
			 
 bResult := BIT_TO_BOOL(stResult.b14_StandByModeActive);
			 
AssertEquals(Expected := bExpected,
             Actual := bResult,
             Message := 'StandByModeActive not set correctly');
			 
bResult := BIT_TO_BOOL(stResult.b15_MovikitHeartbeat);
			 
AssertEquals(Expected := bExpected,
             Actual := bResult,
             Message := 'MovikitHeartbeat not set correctly');
	 
TEST_FINISHED();
END_METHOD

METHOD Test_Cycle_Status_OperationMode : REFERENCE TO FB_Test
VAR_INPUT
	sName 				: T_MaxString;
	bExpected 			: E_SEW_MoviC_Position_OperationMode;
END_VAR

VAR
	fbDrive 			: FB_SEW_MoviC_Position;
	bResult				: E_SEW_MoviC_Position_OperationMode;	
END_VAR
TEST(sName);

fbDrive.stControl.nTargetApplicationMode := bExpected;

fbDrive.Cycle();

bResult := fbDrive.stStatus.nActualApplicationMode;

AssertEquals(Expected := bExpected,
             Actual := bResult,
             Message := 'ApplicationMode not set correctly');
	 
TEST_FINISHED();
END_METHOD

METHOD Test_ProcessDataControl : REFERENCE TO FB_Test
VAR
	fbDrive 						: FB_SEW_MoviC_Position;
	
	nExpectedCW						: WORD;
	nExpectedSetpointSpeed			: INT;
	nExpectedSetpointAcceleration	: INT;
	nExpectedSetpointDeceleration	: INT;
	nExpectedDigitalOutputs			: WORD;
	nExpectedTargetApplicationMode	: E_SEW_MoviC_Position_OperationMode;
	nExpectedTargetPosition			: DINT;
	
	nActualCW						: WORD;
	nActualSetpointSpeed			: INT;
	nActualSetpointAcceleration		: INT;
	nActualSetpointDeceleration		: INT;
	nActualDigitalOutputs			: WORD;
	nActualTargetApplicationMode	: E_SEW_MoviC_Position_OperationMode;
	nActualTargetPosition			: DINT;
		
	stExpectedControlData 		: ST_SEW_MoviC_Position_Control;		
	stActualControlData			: ST_SEW_MoviC_Position_Control;	
END_VAR
TEST('Process data to control structure');

//Arrange
nExpectedCW := 16#A1B2;					
nExpectedSetpointSpeed := UINT_TO_INT(16#C3D4);		
nExpectedSetpointAcceleration := UINT_TO_INT(16#E5F6);		
nExpectedSetpointDeceleration := UINT_TO_INT(16#B6A5);	
nExpectedDigitalOutputs := 16#D4C3;			
nExpectedTargetApplicationMode := 16#F2E1;	
nExpectedTargetPosition := 16#B6A5;

F_Memcpy(ADR(stExpectedControlData), ADR(nExpectedCW), 2, FALSE);
F_Memcpy(ADR(stExpectedControlData) + 2, ADR(nExpectedSetpointSpeed), 2, FALSE);
F_Memcpy(ADR(stExpectedControlData) + 4, ADR(nExpectedSetpointAcceleration), 2, FALSE);
F_Memcpy(ADR(stExpectedControlData) + 6, ADR(nExpectedSetpointDeceleration), 2, FALSE);
F_Memcpy(ADR(stExpectedControlData) + 8, ADR(nExpectedDigitalOutputs), 2, FALSE);
F_Memcpy(ADR(stExpectedControlData) + 10, ADR(nExpectedTargetApplicationMode), 2, FALSE);
F_Memcpy(ADR(stExpectedControlData) + 12, ADR(nExpectedTargetPosition), 4, FALSE);

fbDrive.pControl := ADR(stExpectedControlData);

//Act
fbDrive.GetControlData();

stActualControlData := fbDrive.stControl;

//Assert
F_Memcpy(ADR(nActualCW), ADR(fbDrive.stControl), 2, FALSE);
//F_Memcpy(ADR(nActualTargetVelocity), ADR(fbDrive.stControl) + 2, 2, FALSE);

AssertEquals(Expected := nExpectedCW,
             Actual := nActualCW,
             Message := 'CW is not correct');
	 
AssertEquals(Expected := nExpectedSetpointSpeed,
             Actual := stActualControlData.nSetpointSpeed,
             Message := 'SetpointSpeed is not correct');
			 
AssertEquals(Expected := nExpectedSetpointAcceleration,
             Actual := stActualControlData.nSetpointAcceleration,
             Message := 'SetpointAcceleration is not correct');
			 
AssertEquals(Expected := nExpectedSetpointDeceleration,
             Actual := stActualControlData.nSetpointDeceleration,
             Message := 'SetpointSpeed is not correct');
			 
AssertEquals(Expected := nExpectedDigitalOutputs,
             Actual := stActualControlData.nDigitalOutputs,
             Message := 'SetpointDeceleration is not correct');
			 
AssertEquals(Expected := nExpectedTargetApplicationMode,
             Actual := stActualControlData.nTargetApplicationMode,
             Message := 'TargetApplicationMode is not correct');

AssertEquals(Expected := nExpectedTargetPosition,
             Actual := stActualControlData.nTargetPosition,
             Message := 'TargetPosition is not correct');
			 
TEST_FINISHED();


TEST('Process data to control structure SWAP');

//Arrange
F_Memcpy(ADR(stExpectedControlData), ADR(nExpectedCW), 2, TRUE);
F_Memcpy(ADR(stExpectedControlData) + 2, ADR(nExpectedSetpointSpeed), 2, TRUE);
F_Memcpy(ADR(stExpectedControlData) + 4, ADR(nExpectedSetpointAcceleration), 2, TRUE);
F_Memcpy(ADR(stExpectedControlData) + 6, ADR(nExpectedSetpointDeceleration), 2, TRUE);
F_Memcpy(ADR(stExpectedControlData) + 8, ADR(nExpectedDigitalOutputs), 2, TRUE);
F_Memcpy(ADR(stExpectedControlData) + 10, ADR(nExpectedTargetApplicationMode), 2, TRUE);
F_Memcpy(ADR(stExpectedControlData) + 12, ADR(nExpectedTargetPosition), 4, TRUE);

fbDrive.stConfig.bSwapProcessData := TRUE;

fbDrive.pControl := ADR(stExpectedControlData);

//Act
fbDrive.GetControlData();

stActualControlData := fbDrive.stControl;

//Assert
AssertEquals(Expected := nExpectedCW,
             Actual := nActualCW,
             Message := 'CW is not correct');
	 
AssertEquals(Expected := nExpectedSetpointSpeed,
             Actual := stActualControlData.nSetpointSpeed,
             Message := 'SetpointSpeed is not correct');
			 
AssertEquals(Expected := nExpectedSetpointAcceleration,
             Actual := stActualControlData.nSetpointAcceleration,
             Message := 'SetpointAcceleration is not correct');
			 
AssertEquals(Expected := nExpectedSetpointDeceleration,
             Actual := stActualControlData.nSetpointDeceleration,
             Message := 'SetpointSpeed is not correct');
			 
AssertEquals(Expected := nExpectedDigitalOutputs,
             Actual := stActualControlData.nDigitalOutputs,
             Message := 'SetpointDeceleration is not correct');
			 
AssertEquals(Expected := nExpectedTargetApplicationMode,
             Actual := stActualControlData.nTargetApplicationMode,
             Message := 'TargetApplicationMode is not correct');

AssertEquals(Expected := nExpectedTargetPosition,
             Actual := stActualControlData.nTargetPosition,
             Message := 'TargetPosition is not correct');

TEST_FINISHED();
END_METHOD

METHOD Test_ProcessDataStatus : REFERENCE TO FB_Test
VAR
	fbDrive 						: FB_SEW_MoviC_Position;
	
	nExpectedSW						: WORD;
	nExpectedActualSpeed			: INT;
	nExpectedActualStatus			: WORD;
	nExpectedActualTorque			: INT;
	nExpectedDigitalInputs			: WORD;
	nExpectedActualApplicationMode	: E_SEW_MoviC_Position_OperationMode;
	nExpectedActualPosition			: DINT;
	
	nActualSW						: WORD;
	nActualActualSpeed				: INT;
	nActualActualStatus				: WORD;
	nActualActualTorque				: INT;
	nActualDigitalInputs			: WORD;
	nActualActualApplicationMode	: E_SEW_MoviC_Position_OperationMode;
	nActualActualPosition			: DINT;

	stExpectedStatusData 			: ST_SEW_MoviC_Position_Status;		
	stActualStatusData 				: ST_SEW_MoviC_Position_Status;	
END_VAR
TEST('Assign status structure to process data');

//Arrange
nExpectedSW := 16#A1B2;					
nExpectedActualSpeed := UINT_TO_INT(16#C3D4);		
nExpectedActualStatus := 16#E5F6;		
nExpectedActualTorque := UINT_TO_INT(16#B6A5);	
nExpectedDigitalInputs := 16#B6A5;			
nExpectedActualApplicationMode := UINT_TO_INT(16#B6A5);;	
nExpectedActualPosition := UINT_TO_INT(16#B6A5);;
	
F_Memcpy(ADR(fbDrive.stStatus), ADR(nExpectedSW), 2, FALSE);
F_Memcpy(ADR(fbDrive.stStatus) + 2, ADR(nExpectedActualSpeed), 2, FALSE);
F_Memcpy(ADR(fbDrive.stStatus) + 4, ADR(nExpectedActualStatus), 2, FALSE);
F_Memcpy(ADR(fbDrive.stStatus) + 6, ADR(nExpectedActualTorque), 2, FALSE);
F_Memcpy(ADR(fbDrive.stStatus) + 8, ADR(nExpectedDigitalInputs), 2, FALSE);
F_Memcpy(ADR(fbDrive.stStatus) + 10, ADR(nExpectedActualApplicationMode), 2, FALSE);
F_Memcpy(ADR(fbDrive.stStatus) + 12, ADR(nExpectedActualPosition), 4, FALSE);

fbDrive.pStatus := ADR(stActualStatusData);

//Act
fbDrive.SetStatusData();

//Assert
F_Memcpy(ADR(nActualSW), ADR(stActualStatusData), 2, FALSE);
F_Memcpy(ADR(nActualActualSpeed), ADR(stActualStatusData) + 2, 2, FALSE);
F_Memcpy(ADR(nActualActualStatus), ADR(stActualStatusData) + 4, 2, FALSE);
F_Memcpy(ADR(nActualActualTorque), ADR(stActualStatusData) + 6, 2, FALSE);
F_Memcpy(ADR(nActualDigitalInputs), ADR(stActualStatusData) + 8, 2, FALSE);
F_Memcpy(ADR(nActualActualApplicationMode), ADR(stActualStatusData) + 10, 2, FALSE);
F_Memcpy(ADR(nActualActualPosition), ADR(stActualStatusData)+ 12, 4, FALSE);

AssertEquals(Expected := nExpectedSW,
             Actual := nActualSW,
             Message := 'ZSW1 is not correct');
	 
AssertEquals(Expected := nExpectedActualSpeed,
             Actual := nActualActualSpeed,
             Message := 'ActualVelocity is not correct');	

AssertEquals(Expected := nExpectedActualStatus,
             Actual := nActualActualStatus,
             Message := 'ActualVelocity is not correct');

AssertEquals(Expected := nExpectedActualTorque,
             Actual := nActualActualTorque,
             Message := 'ActualVelocity is not correct');	
				 
AssertEquals(Expected := nExpectedDigitalInputs,
             Actual := nActualDigitalInputs,
             Message := 'ActualVelocity is not correct');	
			 
AssertEquals(Expected := nExpectedActualApplicationMode,
             Actual := nActualActualApplicationMode,
             Message := 'ActualVelocity is not correct');				 
			 
AssertEquals(Expected := nExpectedActualPosition,
             Actual := nActualActualPosition,
             Message := 'ActualVelocity is not correct');				 
			 
TEST_FINISHED();

TEST('Assign status structure to process data SWAP');

//Arrange
nExpectedSW := 16#A1B2;					
nExpectedActualSpeed := UINT_TO_INT(16#C3D4);		
nExpectedActualStatus := 16#E5F6;		
nExpectedActualTorque := UINT_TO_INT(16#B6A5);	
nExpectedDigitalInputs := 16#B6A5;			
nExpectedActualApplicationMode := UINT_TO_INT(16#B6A5);;	
nExpectedActualPosition := UINT_TO_INT(16#B6A5);;
	
F_Memcpy(ADR(fbDrive.stStatus), ADR(nExpectedSW), 2, TRUE);
F_Memcpy(ADR(fbDrive.stStatus) + 2, ADR(nExpectedActualSpeed), 2, TRUE);
F_Memcpy(ADR(fbDrive.stStatus) + 4, ADR(nExpectedActualStatus), 2, TRUE);
F_Memcpy(ADR(fbDrive.stStatus) + 6, ADR(nExpectedActualTorque), 2, TRUE);
F_Memcpy(ADR(fbDrive.stStatus) + 8, ADR(nExpectedDigitalInputs), 2, TRUE);
F_Memcpy(ADR(fbDrive.stStatus) + 10, ADR(nExpectedActualApplicationMode), 2, TRUE);
F_Memcpy(ADR(fbDrive.stStatus) + 12, ADR(nExpectedActualPosition), 4, TRUE);

fbDrive.stConfig.bSwapProcessData := TRUE;

fbDrive.pStatus := ADR(stActualStatusData);

//Act
fbDrive.SetStatusData();

//Assert
F_Memcpy(ADR(nActualSW), ADR(stActualStatusData), 2, FALSE);
F_Memcpy(ADR(nActualActualSpeed), ADR(stActualStatusData) + 2, 2, FALSE);
F_Memcpy(ADR(nActualActualStatus), ADR(stActualStatusData) + 4, 2, FALSE);
F_Memcpy(ADR(nActualActualTorque), ADR(stActualStatusData) + 6, 2, FALSE);
F_Memcpy(ADR(nActualDigitalInputs), ADR(stActualStatusData) + 8, 2, FALSE);
F_Memcpy(ADR(nActualActualApplicationMode), ADR(stActualStatusData) + 10, 2, FALSE);
F_Memcpy(ADR(nActualActualPosition), ADR(stActualStatusData)+ 12, 4, FALSE);

AssertEquals(Expected := nExpectedSW,
             Actual := nActualSW,
             Message := 'ZSW1 is not correct');
	 
AssertEquals(Expected := nExpectedActualSpeed,
             Actual := nActualActualSpeed,
             Message := 'ActualVelocity is not correct');	

AssertEquals(Expected := nExpectedActualStatus,
             Actual := nActualActualStatus,
             Message := 'ActualVelocity is not correct');

AssertEquals(Expected := nExpectedActualTorque,
             Actual := nActualActualTorque,
             Message := 'ActualVelocity is not correct');	
				 
AssertEquals(Expected := nExpectedDigitalInputs,
             Actual := nActualDigitalInputs,
             Message := 'ActualVelocity is not correct');	
			 
AssertEquals(Expected := nExpectedActualApplicationMode,
             Actual := nActualActualApplicationMode,
             Message := 'ActualVelocity is not correct');				 
			 
AssertEquals(Expected := nExpectedActualPosition,
             Actual := nActualActualPosition,
             Message := 'ActualVelocity is not correct');				 
			 
TEST_FINISHED();
END_METHOD

METHOD Test_Safety : REFERENCE TO FB_Test
VAR
	fbDrive 					: FB_SEW_MoviC_Position;
		
	fbSafe						: FB_SEW_Movisafe;
	
	stExpectedSTO				: BOOL;		
	stActualSTO					: BOOL;	
END_VAR
TEST(' Without Safety Interface STO TRUE');

//Arrange
stExpectedSTO := TRUE;
fbDrive.bSTO := stExpectedSTO;

//Act
fbDrive.Safety();

//Assert
stActualSTO := fbDrive.bSTO;

AssertEquals(Expected := stExpectedSTO,
             Actual := stActualSTO,
             Message := 'STO is not correct');
	 		 
TEST_FINISHED();

TEST(' Without Safety Interface STO FALSE');

//Arrange
stExpectedSTO := FALSE;
fbDrive.bSTO := stExpectedSTO;

//Act
fbDrive.Safety();

//Assert
stActualSTO := fbDrive.bSTO;

AssertEquals(Expected := stExpectedSTO,
             Actual := stActualSTO,
             Message := 'STO is not correct');
	 		 
TEST_FINISHED();

TEST('Safety Interface STO TRUE');

//Arrange
stExpectedSTO := TRUE;

fbSafe.bSetSTO := stExpectedSTO;
fbDrive.iMovisafe := fbSafe;

//Act
fbDrive.Safety();

//Assert
stActualSTO := fbDrive.bSTO;

AssertEquals(Expected := stExpectedSTO,
             Actual := stActualSTO,
             Message := 'STO is not correct');
	 		 
TEST_FINISHED();

TEST('Safety Interface FALSE');

//Arrange
stExpectedSTO := FALSE;

fbSafe.bSetSTO := stExpectedSTO;
fbDrive.iMovisafe := fbSafe;

//Act
fbDrive.Safety();

//Assert
stActualSTO := fbDrive.bSTO;

AssertEquals(Expected := stExpectedSTO,
             Actual := stActualSTO,
             Message := 'STO is not correct');
	 		 
TEST_FINISHED();

TEST('Safety Interface false, Overwrite FB input');

//Arrange
stExpectedSTO := FALSE;

fbSafe.bSetSTO := stExpectedSTO;
fbDrive.iMovisafe := fbSafe;
fbDrive.bSTO := NOT stExpectedSTO;

//Act
fbDrive.Safety();

//Assert
stActualSTO := fbDrive.bSTO;

AssertEquals(Expected := stExpectedSTO,
             Actual := stActualSTO,
             Message := 'STO is not correct');
	 		 
TEST_FINISHED();

TEST('Safety Interface true, Overwrite FB input');

//Arrange
stExpectedSTO := TRUE;

fbSafe.bSetSTO := stExpectedSTO;
fbDrive.iMovisafe := fbSafe;
fbDrive.bSTO := NOT stExpectedSTO;

//Act
fbDrive.Safety();

//Assert
stActualSTO := fbDrive.bSTO;

AssertEquals(Expected := stExpectedSTO,
             Actual := stActualSTO,
             Message := 'STO is not correct');
	 		 
TEST_FINISHED();
END_METHOD

END_FUNCTION_BLOCK

// ---- Devices/SEW_MoviC_Position/FB_SEW_MoviC_Position.TcPOU
(*
FB_SEW_MoviC_Position simulates the funcitionalty of a SEW‑EURODRIVE MOVI-C® CONTROLLER with MOVIKIT® Positioning module.

Disclaimer: This simulation is an independent project and is not affiliated with, endorsed by, or approved by SEW‑EURODRIVE. All rights to the SEW‑EURODRIVE brand name and trademarks remain the property of the manufacturer.
Furthermore, no guarantee is given for the completeness of the functional scope or the error-free operation of the simulation. Users should be aware that deviations from the actual product may occur.
*)

{attribute 'reflection'}
FUNCTION_BLOCK FB_SEW_MoviC_Position EXTENDS FB_LinkDataReal
VAR_INPUT
	pControl 			: PVOID; //Pocess data from fieldbus. Size must be >= stControl.
	pStatus 			: PVOID; //Pocess data to fieldbus. Size must be >= stStatus.
	stControl 			: ST_SEW_MoviC_Position_Control; //Control structure. Is read from the fieldbus.
	stConfig 			: ST_SEW_MoviC_Position_Config; //Config structure. Contains parameters of the device.		
	
	bSTO				: BOOL := TRUE;
	iMovisafe			: I_SEW_Movisafe;	
	nDigitalInputs		: WORD;
END_VAR

VAR_OUTPUT
	stStatus			: ST_SEW_MoviC_Position_Status;
	fValue				: REAL;
END_VAR

VAR
    {attribute 'instance-path'} 
    {attribute 'noinit'} 
    _sPath 				: STRING;	                			
	                			
	_fbBaseState		: FB_ProfidriveGSM;
	_fbBasicDrive		: FB_DriveControl;
	                				
	_bOpModeValid		: BOOL;
END_VAR

SUPER^();
InitRun();

GetControlData();
Safety();
Cycle();
SetStatusData();

METHOD INTERNAL Cycle
//Unity Init - Load persistent data
IF SUPER^.Status.7 THEN
	IF stConfig.fRatioPosition <> 0 THEN	
		_fbBasicDrive.fPosition := SUPER^.StatusData/stConfig.fRatioPosition - stConfig.fPositionOffset;
	ELSE
		_fbBasicDrive.fPosition := SUPER^.StatusData - stConfig.fPositionOffset;
	END_IF
END_IF

(* Evaluate incoming operation mode *)
_bOpModeValid := FALSE;

